KUKA KRL program: MyProgram_247().src

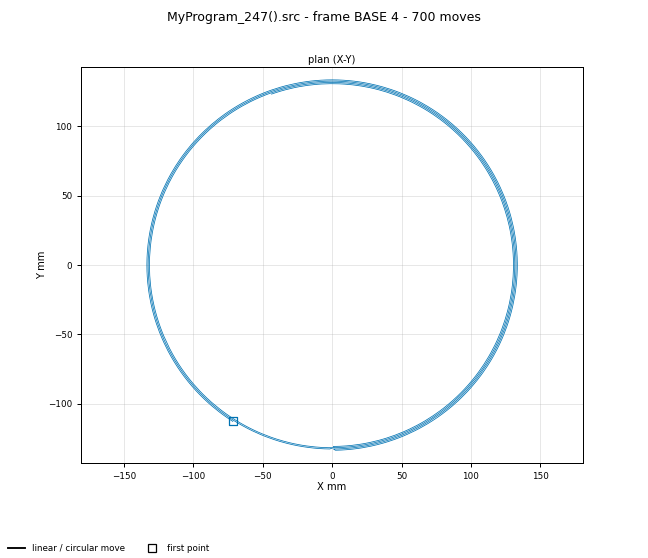
[picture p0: tool path of MyProgram_247().src in frame BASE 4, 700 of 700 moves have a stored position in this frame; points joined in program order, loops and branches not executed]
&ACCESS RVP
&REL 1
&PARAM TEMPLATE = C:\KRC\Roboter\Template\vorgabe
&PARAM EDITMASK = *
DEF MyProgram_247()
; ---- Setting reference (Base) ----
$BASE = BASE_DATA[4]

; --------------------------
; ---- Setting tool (TCP) ----
$TOOL = TOOL_DATA[3]
; --------------------------

$VEL.CP = VEL_APROX_PRINT
Startdeposition()
$VEL.CP = VEL_PRINT
LIN {X -71.493,Y -112.6019,Z 163,A -123.3561,B 17.1544,C -0.1467,E1 17.0685,E2 572.4018} C_DIS
LIN {X -75.0685,Y -110.2504,Z 163,A -125.3445,B 17.1544,C -0.1445,E1 17.0639,E2 574.4076} C_DIS
LIN {X -78.1075,Y -108.1183,Z 163,A -126.8432,B 17.1544,C -0.1504,E1 17.0605,E2 575.894} C_DIS
LIN {X -81.3821,Y -105.6761,Z 163,A -128.5777,B 17.1544,C -0.1541,E1 17.0566,E2 577.6254} C_DIS
LIN {X -86.3277,Y -101.6752,Z 163,A -131.1047,B 17.1542,C -0.166,E1 17.0512,E2 580.1262} C_DIS
LIN {X -88.6867,Y -99.625,Z 163,A -132.7207,B 17.1542,C -0.1593,E1 17.0478,E2 581.7745} C_DIS
LIN {X -91.9669,Y -96.6046,Z 163,A -134.5073,B 17.1542,C -0.1674,E1 17.0442,E2 583.5445} C_DIS
LIN {X -94.7724,Y -93.8538,Z 163,A -136.2946,B 17.1542,C -0.1676,E1 17.0406,E2 585.3427} C_DIS
LIN {X -97.8558,Y -90.6348,Z 163,A -138.7329,B 17.1542,C -0.1544,E1 17.0358,E2 587.8423} C_DIS
LIN {X -100.9904,Y -87.1278,Z 163,A -140.252,B 17.1542,C -0.1754,E1 17.0332,E2 589.3} C_DIS
LIN {X -103.7241,Y -83.8549,Z 163,A -142.1379,B 17.1541,C -0.1777,E1 17.0298,E2 591.1911} C_DIS
LIN {X -106.4808,Y -80.3252,Z 163,A -144.0554,B 17.1541,C -0.1825,E1 17.0265,E2 593.1062} C_DIS
LIN {X -108.9064,Y -77.0047,Z 163,A -145.9648,B 17.1541,C -0.182,E1 17.0234,E2 595.0313} C_DIS
LIN {X -111.3214,Y -73.4702,Z 163,A -147.8571,B 17.1541,C -0.1848,E1 17.0205,E2 596.9283} C_DIS
LIN {X -113.8818,Y -69.4362,Z 163,A -149.7846,B 17.1539,C -0.1941,E1 17.0177,E2 598.8391} C_DIS
LIN {X -116.1067,Y -65.6481,Z 163,A -151.7008,B 17.1539,C -0.198,E1 17.015,E2 600.7569} C_DIS
LIN {X -118.1805,Y -61.8319,Z 163,A -153.4872,B 17.1538,C -0.2055,E1 17.0127,E2 602.5319} C_DIS
LIN {X -121.0994,Y -55.8993,Z 163,A -156.3246,B 17.1537,C -0.2133,E1 17.0092,E2 605.3661} C_DIS
LIN {X -122.6412,Y -52.433,Z 163,A -158.0297,B 17.1537,C -0.2153,E1 17.0073,E2 607.0785} C_DIS
LIN {X -124.4335,Y -48.0231,Z 163,A -160.038,B 17.1536,C -0.2222,E1 17.0052,E2 609.0801} C_DIS
LIN {X -125.5485,Y -45.0269,Z 163,A -161.3821,B 17.1536,C -0.227,E1 17.0039,E2 610.4193} C_DIS
LIN {X -126.5856,Y -42.0228,Z 163,A -162.7229,B 17.1535,C -0.2317,E1 17.0027,E2 611.7555} C_DIS
LIN {X -127.612,Y -38.7951,Z 163,A -164.2281,B 17.1535,C -0.2343,E1 17.0015,E2 613.2651} C_DIS
LIN {X -128.5177,Y -35.6805,Z 163,A -165.6488,B 17.1534,C -0.2375,E1 17.0004,E2 614.6873} C_DIS
LIN {X -129.487,Y -31.9922,Z 163,A -167.8792,B 17.1536,C -0.2233,E1 16.9989,E2 616.986} C_DIS
LIN {X -130.5234,Y -27.4589,Z 163,A -169.4683,B 17.1533,C -0.2423,E1 16.9979,E2 618.5243} C_DIS
LIN {X -131.6134,Y -21.6307,Z 163,A -171.8552,B 17.1531,C -0.2551,E1 16.9968,E2 620.8889} C_DIS
LIN {X -132.1401,Y -18.1495,Z 163,A -174.1734,B 17.1534,C -0.234,E1 16.9959,E2 623.3004} C_DIS
LIN {X -132.774,Y -12.687,Z 163,A -176.0605,B 17.1531,C -0.2562,E1 16.9953,E2 625.1285} C_DIS
LIN {X -133.1204,Y -8.3005,Z 163,A -177.7359,B 17.1529,C -0.2689,E1 16.995,E2 626.7758} C_DIS
LIN {X -133.302,Y -4.5701,Z 163,A -179.3698,B 17.1529,C -0.2728,E1 16.9948,E2 628.4112} C_DIS
LIN {X -133.3812,Y 0.1999,Z 163,A 178.3751,B 17.1529,C -0.2725,E1 16.9948,E2 630.6878} C_DIS
LIN {X -133.2788,Y 5.1658,Z 163,A 176.4508,B 17.1527,C -0.2858,E1 16.9949,E2 632.5843} C_DIS
LIN {X -133.0693,Y 9.1017,Z 163,A 174.457,B 17.1527,C -0.2814,E1 16.9953,E2 634.6113} C_DIS
LIN {X -132.6191,Y 14.2152,Z 163,A 172.1193,B 17.1527,C -0.284,E1 16.9959,E2 636.9614} C_DIS
LIN {X -132.1551,Y 18.0393,Z 163,A 170.7216,B 17.1525,C -0.2972,E1 16.9964,E2 638.3265} C_DIS
LIN {X -131.5675,Y 21.906,Z 163,A 169.1689,B 17.1523,C -0.3064,E1 16.9971,E2 639.8618} C_DIS
LIN {X -130.991,Y 25.1241,Z 163,A 167.6851,B 17.1523,C -0.3081,E1 16.9979,E2 641.3529} C_DIS
LIN {X -129.9919,Y 29.8659,Z 163,A 165.6622,B 17.1521,C -0.3163,E1 16.9991,E2 643.3658} C_DIS
LIN {X -129.2337,Y 32.993,Z 163,A 164.2204,B 17.1521,C -0.3186,E1 17,E2 644.8127} C_DIS
LIN {X -127.6785,Y 38.578,Z 163,A 161.5292,B 17.1521,C -0.3196,E1 17.0021,E2 647.524} C_DIS
LIN {X -126.4721,Y 42.3638,Z 163,A 159.979,B 17.1519,C -0.3297,E1 17.0035,E2 649.0532} C_DIS
LIN {X -125.1164,Y 46.2174,Z 163,A 158.1128,B 17.1519,C -0.3312,E1 17.0052,E2 650.93} C_DIS
LIN {X -122.6784,Y 52.3471,Z 163,A 155.4199,B 17.1516,C -0.344,E1 17.008,E2 653.6022} C_DIS
LIN {X -121.5681,Y 54.8744,Z 163,A 154.0171,B 17.1516,C -0.3404,E1 17.0097,E2 655.0289} C_DIS
LIN {X -118.3417,Y 61.5248,Z 163,A 151.085,B 17.1514,C -0.3571,E1 17.0133,E2 657.9277} C_DIS
LIN {X -116.0256,Y 65.7912,Z 163,A 148.7366,B 17.1514,C -0.3544,E1 17.0164,E2 660.3042} C_DIS
LIN {X -112.7569,Y 71.2474,Z 163,A 146.0518,B 17.1512,C -0.3632,E1 17.0203,E2 662.9795} C_DIS
LIN {X -109.7743,Y 75.763,Z 163,A 143.9098,B 17.151,C -0.3752,E1 17.0236,E2 665.0967} C_DIS
LIN {X -107.8305,Y 78.5046,Z 163,A 142.287,B 17.151,C -0.3731,E1 17.0263,E2 666.7386} C_DIS
LIN {X -105.2804,Y 81.8925,Z 163,A 140.2017,B 17.1511,C -0.3692,E1 17.0299,E2 668.8525} C_DIS
LIN {X -101.3359,Y 86.7267,Z 163,A 137.9244,B 17.1507,C -0.3888,E1 17.0339,E2 671.0787} C_DIS
LIN {X -99.1859,Y 89.177,Z 163,A 135.6773,B 17.1512,C -0.3647,E1 17.0382,E2 673.4232} C_DIS
LIN {X -95.5933,Y 93.018,Z 163,A 133.3776,B 17.1512,C -0.3686,E1 17.0427,E2 675.7246} C_DIS
LIN {X -91.7673,Y 96.7945,Z 163,A 131.9655,B 17.1504,C -0.4029,E1 17.0453,E2 677.0286} C_DIS
LIN {X -86.6154,Y 101.4291,Z 163,A 128.4729,B 17.1506,C -0.3923,E1 17.0527,E2 680.5781} C_DIS
LIN {X -84.0592,Y 103.5591,Z 163,A 127.3266,B 17.1503,C -0.4045,E1 17.0551,E2 681.6894} C_DIS
LIN {X -81.7259,Y 105.4096,Z 163,A 125.9695,B 17.1503,C -0.4045,E1 17.0581,E2 683.0541} C_DIS
LIN {X -77.298,Y 108.6989,Z 163,A 123.7781,B 17.1501,C -0.4149,E1 17.063,E2 685.2217} C_DIS
LIN {X -74.477,Y 110.6508,Z 163,A 122.1784,B 17.1501,C -0.4134,E1 17.0667,E2 686.8346} C_DIS
LIN {X -71.3132,Y 112.7154,Z 163,A 120.5812,B 17.1501,C -0.4171,E1 17.0705,E2 688.4269} C_DIS
LIN {X -68.2373,Y 114.6036,Z 163,A 118.9103,B 17.1501,C -0.4157,E1 17.0745,E2 690.1103} C_DIS
LIN {X -64.4041,Y 116.801,Z 163,A 116.4812,B 17.1504,C -0.4012,E1 17.0806,E2 692.5995} C_DIS
LIN {X -60.2581,Y 118.9908,Z 163,A 114.7353,B 17.1501,C -0.4131,E1 17.0848,E2 694.3119} C_DIS
LIN {X -57.2362,Y 120.4736,Z 163,A 113.5999,B 17.1499,C -0.4256,E1 17.0876,E2 695.4093} C_DIS
LIN {X -53.7854,Y 122.0552,Z 163,A 111.6553,B 17.1501,C -0.4172,E1 17.0926,E2 697.3892} C_DIS
LIN {X -50.7486,Y 123.3486,Z 163,A 110.43,B 17.1499,C -0.4255,E1 17.0957,E2 698.5906} C_DIS
LIN {X -46.8423,Y 124.8824,Z 163,A 108.7335,B 17.1497,C -0.4313,E1 17.1001,E2 700.2728} C_DIS
LIN {X -43.603,Y 126.05,Z 163,A 106.2735,B 17.1504,C -0.4,E1 17.1069,E2 702.8461} C_DIS
LIN {X -37.145,Y 128.1023,Z 163,A 104.3419,B 17.1496,C -0.4359,E1 17.1118,E2 704.6608} C_DIS
LIN {X -33.258,Y 129.1664,Z 163,A 102.5415,B 17.1496,C -0.4351,E1 17.1166,E2 706.4681} C_DIS
LIN {X -26.3839,Y 130.7432,Z 163,A 99.5247,B 17.1496,C -0.4379,E1 17.1249,E2 709.481} C_DIS
LIN {X -22.6279,Y 131.447,Z 163,A 97.7835,B 17.1496,C -0.4355,E1 17.1297,E2 711.2328} C_DIS
LIN {X -18.8702,Y 132.0371,Z 163,A 96.2962,B 17.1495,C -0.4415,E1 17.1337,E2 712.7017} C_DIS
LIN {X -15.3622,Y 132.4918,Z 163,A 94.7327,B 17.1495,C -0.4407,E1 17.1381,E2 714.2695} C_DIS
LIN {X -11.4017,Y 132.8907,Z 163,A 93.0376,B 17.1495,C -0.4419,E1 17.1428,E2 715.9617} C_DIS
LIN {X -8.1027,Y 133.1325,Z 163,A 91.61,B 17.1495,C -0.4422,E1 17.1468,E2 717.3892} C_DIS
LIN {X -4.0439,Y 133.318,Z 163,A 89.8115,B 17.1495,C -0.4407,E1 17.1518,E2 719.1932} C_DIS
LIN {X 0.0154,Y 133.3809,Z 163,A 87.9798,B 17.1495,C -0.4379,E1 17.1569,E2 721.0344} C_DIS
LIN {X 4.194,Y 133.3138,Z 163,A 86.2031,B 17.1495,C -0.4386,E1 17.1619,E2 722.808} C_DIS
LIN {X 8.2626,Y 133.1227,Z 163,A 84.6014,B 17.1495,C -0.4437,E1 17.1663,E2 724.3916} C_DIS
LIN {X 11.8743,Y 132.8508,Z 163,A 82.8734,B 17.1495,C -0.4374,E1 17.1712,E2 726.1393} C_DIS
LIN {X 15.9022,Y 132.4274,Z 163,A 81.2741,B 17.1495,C -0.442,E1 17.1756,E2 727.7215} C_DIS
LIN {X 19.7309,Y 131.913,Z 163,A 79.5121,B 17.1495,C -0.4379,E1 17.1805,E2 729.4952} C_DIS
LIN {X 23.404,Y 131.3093,Z 163,A 78.0206,B 17.1495,C -0.441,E1 17.1845,E2 730.9734} C_DIS
LIN {X 26.981,Y 130.6217,Z 163,A 75.7507,B 17.1501,C -0.4153,E1 17.191,E2 733.3263} C_DIS
LIN {X 32.3107,Y 129.4068,Z 163,A 74.2533,B 17.1494,C -0.4441,E1 17.1948,E2 734.7229} C_DIS
LIN {X 36.0725,Y 128.4081,Z 163,A 72.4271,B 17.1496,C -0.4374,E1 17.1997,E2 736.5672} C_DIS
LIN {X 39.3278,Y 127.449,Z 163,A 70.9977,B 17.1496,C -0.4373,E1 17.2035,E2 737.9932} C_DIS
LIN {X 42.3688,Y 126.4704,Z 163,A 69.6413,B 17.1496,C -0.4367,E1 17.2071,E2 739.3476} C_DIS
LIN {X 45.6944,Y 125.3079,Z 163,A 68.1255,B 17.1496,C -0.4352,E1 17.2111,E2 740.8637} C_DIS
LIN {X 48.7199,Y 124.1626,Z 163,A 66.75,B 17.1496,C -0.4344,E1 17.2147,E2 742.2377} C_DIS
LIN {X 51.816,Y 122.9028,Z 163,A 65.3241,B 17.1496,C -0.4332,E1 17.2184,E2 743.6624} C_DIS
LIN {X 54.7217,Y 121.6364,Z 163,A 63.954,B 17.1497,C -0.4313,E1 17.2219,E2 745.0337} C_DIS
LIN {X 57.9536,Y 120.1308,Z 163,A 62.3008,B 17.1499,C -0.4251,E1 17.2261,E2 746.7017} C_DIS
LIN {X 61.1871,Y 118.5179,Z 163,A 60.8946,B 17.1498,C -0.4284,E1 17.2295,E2 748.0908} C_DIS
LIN {X 63.9805,Y 117.0334,Z 163,A 59.243,B 17.1501,C -0.4158,E1 17.2337,E2 749.7776} C_DIS
LIN {X 68.7879,Y 114.2743,Z 163,A 57.0624,B 17.15,C -0.4197,E1 17.2389,E2 751.9351} C_DIS
LIN {X 72.4699,Y 111.9753,Z 163,A 55.1281,B 17.1501,C -0.4143,E1 17.2435,E2 753.8782} C_DIS
LIN {X 76.0879,Y 109.5488,Z 163,A 53.3455,B 17.1501,C -0.4145,E1 17.2475,E2 755.6509} C_DIS
LIN {X 79.6618,Y 106.9781,Z 163,A 51.4591,B 17.1501,C -0.4114,E1 17.2518,E2 757.5375} C_DIS
LIN {X 83.2162,Y 104.2372,Z 163,A 49.5443,B 17.1503,C -0.4084,E1 17.256,E2 759.4516} C_DIS
LIN {X 86.6973,Y 101.361,Z 163,A 47.5814,B 17.1503,C -0.4039,E1 17.2602,E2 761.4184} C_DIS
LIN {X 90.0715,Y 98.3743,Z 163,A 45.6822,B 17.1504,C -0.4015,E1 17.2641,E2 763.3142} C_DIS
LIN {X 93.2865,Y 95.3308,Z 163,A 43.8058,B 17.1504,C -0.3985,E1 17.2679,E2 765.1888} C_DIS
LIN {X 96.3446,Y 92.2391,Z 163,A 41.9487,B 17.1506,C -0.395,E1 17.2715,E2 767.0458} C_DIS
LIN {X 99.4016,Y 88.9361,Z 163,A 40.0407,B 17.1506,C -0.3917,E1 17.2751,E2 768.952} C_DIS
LIN {X 102.3672,Y 85.5064,Z 163,A 38.0904,B 17.1507,C -0.3872,E1 17.2787,E2 770.9041} C_DIS
LIN {X 105.1727,Y 82.0315,Z 163,A 36.1803,B 17.1508,C -0.3831,E1 17.282,E2 772.8147} C_DIS
LIN {X 108.0905,Y 78.1459,Z 163,A 34.3877,B 17.1507,C -0.3893,E1 17.2849,E2 774.5736} C_DIS
LIN {X 109.735,Y 75.8203,Z 163,A 32.8867,B 17.151,C -0.3757,E1 17.2874,E2 776.1091} C_DIS
LIN {X 112.1364,Y 72.221,Z 163,A 31.0231,B 17.151,C -0.3709,E1 17.2902,E2 777.9748} C_DIS
LIN {X 114.4652,Y 68.4695,Z 163,A 29.1486,B 17.1512,C -0.3669,E1 17.2929,E2 779.8483} C_DIS
LIN {X 116.6388,Y 64.6972,Z 163,A 27.3166,B 17.1512,C -0.3635,E1 17.2954,E2 781.6776} C_DIS
LIN {X 119.3725,Y 59.4986,Z 163,A 24.755,B 17.1514,C -0.3553,E1 17.2987,E2 784.2463} C_DIS
LIN {X 121.0966,Y 55.9054,Z 163,A 23.2334,B 17.1514,C -0.3579,E1 17.3005,E2 785.7466} C_DIS
LIN {X 122.475,Y 52.8174,Z 163,A 21.768,B 17.1514,C -0.3534,E1 17.3022,E2 787.2152} C_DIS
LIN {X 123.7138,Y 49.8466,Z 163,A 20.3661,B 17.1515,C -0.3488,E1 17.3037,E2 788.6209} C_DIS
LIN {X 125.0163,Y 46.4848,Z 163,A 18.8361,B 17.1516,C -0.3451,E1 17.3052,E2 790.1504} C_DIS
LIN {X 126.7022,Y 41.6726,Z 163,A 16.4693,B 17.1519,C -0.3321,E1 17.3073,E2 792.5411} C_DIS
LIN {X 127.9499,Y 37.6655,Z 163,A 14.8838,B 17.1518,C -0.3352,E1 17.3086,E2 794.1024} C_DIS
LIN {X 128.8888,Y 34.3151,Z 163,A 13.3791,B 17.1518,C -0.3304,E1 17.3097,E2 795.6101} C_DIS
LIN {X 130.5446,Y 27.3602,Z 163,A 10.4004,B 17.152,C -0.3248,E1 17.3116,E2 798.5815} C_DIS
LIN {X 131.0616,Y 24.7551,Z 163,A 9.1989,B 17.152,C -0.3191,E1 17.3122,E2 799.7917} C_DIS
LIN {X 131.8029,Y 20.4418,Z 163,A 7.3681,B 17.1522,C -0.3153,E1 17.313,E2 801.619} C_DIS
LIN {X 132.2935,Y 16.9835,Z 163,A 5.9213,B 17.1522,C -0.3129,E1 17.3136,E2 803.0612} C_DIS
LIN {X 132.7376,Y 13.0661,Z 163,A 4.1856,B 17.1523,C -0.3061,E1 17.3141,E2 804.8042} C_DIS
LIN {X 133.0365,Y 9.5509,Z 163,A 2.7026,B 17.1523,C -0.3027,E1 17.3144,E2 806.2854} C_DIS
LIN {X 133.2713,Y 5.3591,Z 163,A 0.8516,B 17.1525,C -0.2953,E1 17.3147,E2 808.1446} C_DIS
LIN {X 133.3772,Y 0.8301,Z 163,A -0.9648,B 17.1525,C -0.2944,E1 17.3147,E2 809.9479} C_DIS
LIN {X 133.3491,Y -2.9015,Z 163,A -2.7829,B 17.1527,C -0.2811,E1 17.3147,E2 811.7944} C_DIS
LIN {X 133.172,Y -7.462,Z 163,A -4.6776,B 17.1527,C -0.2776,E1 17.3144,E2 813.6838} C_DIS
LIN {X 132.8946,Y -11.3554,Z 163,A -6.2039,B 17.1527,C -0.2783,E1 17.3141,E2 815.1942} C_DIS
LIN {X 132.5722,Y -14.651,Z 163,A -7.5931,B 17.1528,C -0.2752,E1 17.3137,E2 816.5814} C_DIS
LIN {X 132.0755,Y -18.6012,Z 163,A -9.3503,B 17.1529,C -0.2681,E1 17.3131,E2 818.3467} C_DIS
LIN {X 131.491,Y -22.3645,Z 163,A -10.9245,B 17.1529,C -0.2655,E1 17.3124,E2 819.9157} C_DIS
LIN {X 130.0759,Y -29.4984,Z 163,A -13.7711,B 17.1529,C -0.2668,E1 17.3108,E2 822.733} C_DIS
LIN {X 129.0527,Y -33.7004,Z 163,A -15.95,B 17.1532,C -0.2487,E1 17.3093,E2 824.9539} C_DIS
LIN {X 128.0391,Y -37.361,Z 163,A -17.5537,B 17.1532,C -0.2449,E1 17.3081,E2 826.5565} C_DIS
LIN {X 126.9864,Y -40.796,Z 163,A -18.9769,B 17.1532,C -0.2449,E1 17.3069,E2 827.9674} C_DIS
LIN {X 125.9675,Y -43.8408,Z 163,A -20.3842,B 17.1533,C -0.2398,E1 17.3056,E2 829.38} C_DIS
LIN {X 124.826,Y -46.9928,Z 163,A -21.7511,B 17.1533,C -0.2384,E1 17.3043,E2 830.7402} C_DIS
LIN {X 123.6614,Y -49.9767,Z 163,A -23.1582,B 17.1534,C -0.2331,E1 17.3029,E2 832.1531} C_DIS
LIN {X 122.3286,Y -53.156,Z 163,A -24.6723,B 17.1535,C -0.2276,E1 17.3012,E2 833.6734} C_DIS
LIN {X 120.529,Y -57.1202,Z 163,A -26.973,B 17.1538,C -0.2056,E1 17.2984,E2 836.0292} C_DIS
LIN {X 118.6252,Y -60.9763,Z 163,A -28.1414,B 17.1535,C -0.2266,E1 17.297,E2 837.1176} C_DIS
LIN {X 116.3629,Y -65.1922,Z 163,A -30.2966,B 17.1536,C -0.217,E1 17.2942,E2 839.2881} C_DIS
LIN {X 114.4383,Y -68.5147,Z 163,A -32.0816,B 17.1538,C -0.2072,E1 17.2916,E2 841.0921} C_DIS
LIN {X 111.9838,Y -72.4567,Z 163,A -34.7078,B 17.1541,C -0.1777,E1 17.2875,E2 843.7977} C_DIS
LIN {X 108.8457,Y -77.0908,Z 163,A -36.1924,B 17.1538,C -0.2066,E1 17.2853,E2 845.174} C_DIS
LIN {X 107.0794,Y -79.5257,Z 163,A -38.1888,B 17.1541,C -0.1763,E1 17.2819,E2 847.258} C_DIS
LIN {X 104.2672,Y -83.1786,Z 163,A -39.7653,B 17.154,C -0.1868,E1 17.2792,E2 848.7882} C_DIS
LIN {X 100.1471,Y -88.0963,Z 163,A -42.449,B 17.154,C -0.1828,E1 17.2743,E2 851.4669} C_DIS
LIN {X 97.187,Y -91.3512,Z 163,A -44.3323,B 17.154,C -0.1785,E1 17.2708,E2 853.352} C_DIS
LIN {X 93.0583,Y -95.5538,Z 163,A -47.0279,B 17.1542,C -0.1665,E1 17.2654,E2 856.071} C_DIS
LIN {X 90.6712,Y -97.822,Z 163,A -47.9557,B 17.154,C -0.1819,E1 17.2636,E2 856.9411} C_DIS
LIN {X 86.8093,Y -101.2647,Z 163,A -50.4464,B 17.1542,C -0.1669,E1 17.2583,E2 859.4675} C_DIS
LIN {X 82.6931,Y -104.6526,Z 163,A -53.1213,B 17.1544,C -0.1476,E1 17.2524,E2 862.1921} C_DIS
LIN {X 79.2187,Y -107.3071,Z 163,A -54.5595,B 17.1542,C -0.1605,E1 17.2493,E2 863.5792} C_DIS
LIN {X 75.7434,Y -109.7877,Z 163,A -56.7712,B 17.1544,C -0.1428,E1 17.2441,E2 865.839} C_DIS
LIN {X 72.302,Y -112.084,Z 163,A -58.1844,B 17.1544,C -0.1532,E1 17.2409,E2 867.21} C_DIS
LIN {X 68.6071,Y -114.3832,Z 163,A -60.018,B 17.1544,C -0.1513,E1 17.2365,E2 869.0414} C_DIS
LIN {X 63.2632,Y -117.4228,Z 163,A -62.6363,B 17.1544,C -0.1478,E1 17.2302,E2 871.6597} C_DIS
LIN {X 59.8567,Y -119.1952,Z 163,A -64.5342,B 17.1544,C -0.136,E1 17.2254,E2 873.5897} C_DIS
LIN {X 56.7284,Y -120.716,Z 163,A -65.6812,B 17.1544,C -0.1467,E1 17.2226,E2 874.6959} C_DIS
LIN {X 54.1774,Y -121.8798,Z 163,A -66.8721,B 17.1544,C -0.1455,E1 17.2195,E2 875.8863} C_DIS
LIN {X 51.3383,Y -123.1023,Z 163,A -68.2057,B 17.1544,C -0.1435,E1 17.2161,E2 877.2219} C_DIS
LIN {X 48.1656,Y -124.3781,Z 163,A -69.714,B 17.1544,C -0.1402,E1 17.2122,E2 878.7365} C_DIS
LIN {X 44.5567,Y -125.7181,Z 163,A -71.4591,B 17.1544,C -0.1348,E1 17.2076,E2 880.4943} C_DIS
LIN {X 39.6414,Y -127.353,Z 163,A -73.543,B 17.1544,C -0.1375,E1 17.2021,E2 882.563} C_DIS
LIN {X 36.5954,Y -128.2618,Z 163,A -75.4292,B 17.1546,C -0.117,E1 17.1968,E2 884.5136} C_DIS
LIN {X 32.3464,Y -129.3978,Z 163,A -76.8995,B 17.1545,C -0.1306,E1 17.193,E2 885.9346} C_DIS
LIN {X 28.253,Y -130.352,Z 163,A -78.6338,B 17.1545,C -0.1317,E1 17.1883,E2 887.6617} C_DIS
LIN {X 24.7601,Y -131.0606,Z 163,A -80.1063,B 17.1545,C -0.1327,E1 17.1842,E2 889.1282} C_DIS
LIN {X 21.814,Y -131.5828,Z 163,A -81.396,B 17.1545,C -0.1316,E1 17.1807,E2 890.4193} C_DIS
LIN {X 18.6748,Y -132.065,Z 163,A -82.7582,B 17.1545,C -0.1309,E1 17.1769,E2 891.7821} C_DIS
LIN {X 14.6266,Y -132.5748,Z 163,A -84.5987,B 17.1545,C -0.1268,E1 17.1718,E2 893.6346} C_DIS
LIN {X 10.5342,Y -132.964,Z 163,A -86.4015,B 17.1545,C -0.1246,E1 17.1668,E2 895.443} C_DIS
LIN {X 6.5935,Y -133.2158,Z 163,A -87.9976,B 17.1545,C -0.1277,E1 17.1623,E2 897.0278} C_DIS
LIN {X 2.3994,Y -133.3575,Z 163,A -89.8236,B 17.1545,C -0.1264,E1 17.1572,E2 898.8576} C_DIS
LIN {X 2.3994,Y -133.3575,Z 163,A -89.8236,B 17.1545,C -0.1264,E1 17.1572,E2 898.8576} C_DIS
Enddeposition()
LIN {X 0.9252,Y -132.4528,Z 163,A -88.4816,B 12.714,C 0.1927,E1 12.718,E2 898.6293} C_DIS
Startdeposition()
$VEL.CP = VEL_PRINT
LIN {X 4.65,Y -132.3773,Z 163,A -86.7032,B 12.714,C 0.1879,E1 12.7231,E2 896.8298} C_DIS
LIN {X 8.6149,Y -132.1783,Z 163,A -84.9273,B 12.714,C 0.1858,E1 12.728,E2 895.0459} C_DIS
LIN {X 13.043,Y -131.8147,Z 163,A -83.1114,B 12.714,C 0.1879,E1 12.7331,E2 893.2417} C_DIS
LIN {X 16.933,Y -131.3713,Z 163,A -81.3857,B 12.714,C 0.1862,E1 12.7379,E2 891.5112} C_DIS
LIN {X 20.7774,Y -130.8191,Z 163,A -79.6446,B 12.7141,C 0.1835,E1 12.7427,E2 889.7615} C_DIS
LIN {X 24.735,Y -130.1278,Z 163,A -78.0449,B 12.7141,C 0.1861,E1 12.747,E2 888.1775} C_DIS
LIN {X 27.8978,Y -129.4865,Z 163,A -76.6131,B 12.7141,C 0.1841,E1 12.751,E2 886.7403} C_DIS
LIN {X 31.8651,Y -128.5698,Z 163,A -74.1973,B 12.7144,C 0.1644,E1 12.7578,E2 884.2427} C_DIS
LIN {X 36.8579,Y -127.2268,Z 163,A -72.8328,B 12.7141,C 0.1866,E1 12.7611,E2 882.9837} C_DIS
LIN {X 40.5932,Y -126.0845,Z 163,A -70.9607,B 12.7141,C 0.1798,E1 12.7662,E2 881.088} C_DIS
LIN {X 44.0819,Y -124.9093,Z 163,A -69.292,B 12.7142,C 0.176,E1 12.7706,E2 879.4087} C_DIS
LIN {X 48.0926,Y -123.4184,Z 163,A -67.5243,B 12.7142,C 0.176,E1 12.7752,E2 877.6495} C_DIS
LIN {X 51.8287,Y -121.8992,Z 163,A -65.7247,B 12.7142,C 0.1723,E1 12.7799,E2 875.8418} C_DIS
LIN {X 55.3976,Y -120.3168,Z 163,A -64.3685,B 12.7142,C 0.1794,E1 12.7832,E2 874.5246} C_DIS
LIN {X 61.0215,Y -117.5659,Z 163,A -60.6564,B 12.7146,C 0.1469,E1 12.7928,E2 870.6866} C_DIS
LIN {X 66.1056,Y -114.7852,Z 163,A -58.8364,B 12.7144,C 0.1627,E1 12.797,E2 868.949} C_DIS
LIN {X 69.5157,Y -112.7526,Z 163,A -57.1776,B 12.7144,C 0.1615,E1 12.801,E2 867.2957} C_DIS
LIN {X 77.6184,Y -107.3354,Z 163,A -52.9856,B 12.7144,C 0.1547,E1 12.8107,E2 863.1026} C_DIS
LIN {X 79.9123,Y -105.6387,Z 163,A -51.4002,B 12.7146,C 0.1422,E1 12.8143,E2 861.4726} C_DIS
LIN {X 83.0042,Y -103.2271,Z 163,A -50.2306,B 12.7145,C 0.1542,E1 12.8167,E2 860.366} C_DIS
LIN {X 86.6021,Y -100.2278,Z 163,A -48.0441,B 12.7145,C 0.1454,E1 12.8214,E2 858.1576} C_DIS
LIN {X 89.442,Y -97.7021,Z 163,A -45.8817,B 12.7148,C 0.1269,E1 12.826,E2 855.9296} C_DIS
LIN {X 93.0322,Y -94.29,Z 163,A -44.3094,B 12.7147,C 0.1389,E1 12.829,E2 854.4252} C_DIS
LIN {X 96.812,Y -90.4044,Z 163,A -41.9462,B 12.7147,C 0.1331,E1 12.8336,E2 852.0571} C_DIS
LIN {X 99.0129,Y -87.9889,Z 163,A -39.868,B 12.7149,C 0.1103,E1 12.8376,E2 849.8952} C_DIS
LIN {X 102.7772,Y -83.561,Z 163,A -38.3365,B 12.7147,C 0.1333,E1 12.8401,E2 848.4819} C_DIS
LIN {X 104.5434,Y -81.3394,Z 163,A -36.5214,B 12.7149,C 0.113,E1 12.8433,E2 846.5932} C_DIS
LIN {X 106.9368,Y -78.1672,Z 163,A -35.1598,B 12.7149,C 0.1193,E1 12.8455,E2 845.2735} C_DIS
LIN {X 111.7951,Y -71.0459,Z 163,A -31.4795,B 12.7149,C 0.1114,E1 12.8512,E2 841.5949} C_DIS
LIN {X 114.0314,Y -67.3978,Z 163,A -29.6337,B 12.7149,C 0.1067,E1 12.8539,E2 839.7475} C_DIS
LIN {X 115.9202,Y -64.0937,Z 163,A -27.7268,B 12.7151,C 0.0946,E1 12.8565,E2 837.8066} C_DIS
LIN {X 117.6362,Y -60.8876,Z 163,A -26.5258,B 12.7151,C 0.1014,E1 12.858,E2 836.6493} C_DIS
LIN {X 120.0623,Y -55.9478,Z 163,A -24.1864,B 12.7151,C 0.0961,E1 12.8609,E2 834.3121} C_DIS
LIN {X 121.4879,Y -52.78,Z 163,A -22.7613,B 12.7151,C 0.0942,E1 12.8625,E2 832.8946} C_DIS
LIN {X 122.7392,Y -49.8012,Z 163,A -21.4109,B 12.7151,C 0.0917,E1 12.8639,E2 831.5482} C_DIS
LIN {X 123.8897,Y -46.867,Z 163,A -19.9341,B 12.7151,C 0.0845,E1 12.8654,E2 830.0559} C_DIS
LIN {X 125.0887,Y -43.5644,Z 163,A -18.4302,B 12.7151,C 0.0807,E1 12.8668,E2 828.5522} C_DIS
LIN {X 126.1966,Y -40.2422,Z 163,A -16.9364,B 12.7151,C 0.077,E1 12.8681,E2 827.0591} C_DIS
LIN {X 127.3419,Y -36.4623,Z 163,A -15.1507,B 12.7152,C 0.0697,E1 12.8695,E2 825.2619} C_DIS
LIN {X 128.351,Y -32.7272,Z 163,A -13.6612,B 12.7152,C 0.0704,E1 12.8705,E2 823.7928} C_DIS
LIN {X 129.8568,Y -26.1202,Z 163,A -10.7284,B 12.7152,C 0.0618,E1 12.8723,E2 820.8565} C_DIS
LIN {X 130.6013,Y -22.1011,Z 163,A -8.9604,B 12.7152,C 0.0566,E1 12.8732,E2 819.0863} C_DIS
LIN {X 131.1939,Y -18.2611,Z 163,A -7.1977,B 12.7153,C 0.0491,E1 12.8739,E2 817.3117} C_DIS
LIN {X 131.7029,Y -14.1219,Z 163,A -5.5797,B 12.7153,C 0.0493,E1 12.8744,E2 815.7142} C_DIS
LIN {X 132.0106,Y -10.8795,Z 163,A -4.043,B 12.7153,C 0.0413,E1 12.8748,E2 814.1604} C_DIS
LIN {X 132.2761,Y -6.9447,Z 163,A -2.4321,B 12.7153,C 0.0391,E1 12.875,E2 812.559} C_DIS
LIN {X 132.4304,Y -2.7627,Z 163,A -0.5578,B 12.7153,C 0.0318,E1 12.8752,E2 810.6749} C_DIS
LIN {X 132.4517,Y 1.4833,Z 163,A 1.296,B 12.7153,C 0.0259,E1 12.8752,E2 808.817} C_DIS
LIN {X 132.3361,Y 5.7074,Z 163,A 3.0736,B 12.7153,C 0.0219,E1 12.875,E2 807.0435} C_DIS
LIN {X 132.0915,Y 9.848,Z 163,A 4.7989,B 12.7153,C 0.0187,E1 12.8747,E2 805.3246} C_DIS
LIN {X 131.7124,Y 14.0336,Z 163,A 6.4926,B 12.7153,C 0.017,E1 12.8742,E2 803.644} C_DIS
LIN {X 131.3276,Y 17.2665,Z 163,A 7.8923,B 12.7153,C 0.0131,E1 12.8737,E2 802.2439} C_DIS
LIN {X 130.8393,Y 20.6471,Z 163,A 9.4762,B 12.7154,C 0.0056,E1 12.873,E2 800.6456} C_DIS
LIN {X 130.1395,Y 24.6741,Z 163,A 11.1431,B 12.7154,C 0.0035,E1 12.8722,E2 798.9891} C_DIS
LIN {X 128.3566,Y 32.7051,Z 163,A 14.7923,B 12.7154,C -0.0094,E1 12.8699,E2 795.3256} C_DIS
LIN {X 126.9678,Y 37.7421,Z 163,A 17.7638,B 12.7154,C -0.0369,E1 12.8675,E2 792.2652} C_DIS
LIN {X 125.0134,Y 43.7817,Z 163,A 19.7259,B 12.7154,C -0.0213,E1 12.8658,E2 790.3963} C_DIS
LIN {X 123.5745,Y 47.691,Z 163,A 21.4127,B 12.7154,C -0.0228,E1 12.8642,E2 788.7218} C_DIS
LIN {X 122.2595,Y 50.9666,Z 163,A 22.8699,B 12.7154,C -0.0249,E1 12.8626,E2 787.2717} C_DIS
LIN {X 120.8602,Y 54.2016,Z 163,A 24.3713,B 12.7154,C -0.0283,E1 12.8609,E2 785.7718} C_DIS
LIN {X 119.7096,Y 56.6991,Z 163,A 26.0355,B 12.7154,C -0.0454,E1 12.8589,E2 784.0493} C_DIS
LIN {X 117.8824,Y 60.4055,Z 163,A 27.4023,B 12.7154,C -0.0377,E1 12.8572,E2 782.732} C_DIS
LIN {X 115.6998,Y 64.4917,Z 163,A 29.396,B 12.7154,C -0.0426,E1 12.8545,E2 780.7381} C_DIS
LIN {X 113.8882,Y 67.6389,Z 163,A 30.9874,B 12.7154,C -0.0471,E1 12.8523,E2 779.1431} C_DIS
LIN {X 111.4568,Y 71.5744,Z 163,A 32.8954,B 12.7154,C -0.0494,E1 12.8495,E2 777.2449} C_DIS
LIN {X 109.5164,Y 74.51,Z 163,A 34.4599,B 12.7153,C -0.0543,E1 12.847,E2 775.6743} C_DIS
LIN {X 106.961,Y 78.1334,Z 163,A 36.3454,B 12.7153,C -0.0579,E1 12.844,E2 773.7914} C_DIS
LIN {X 104.3973,Y 81.5281,Z 163,A 38.1939,B 12.7153,C -0.0623,E1 12.8408,E2 771.9409} C_DIS
LIN {X 101.7273,Y 84.8364,Z 163,A 40.0347,B 12.7153,C -0.0665,E1 12.8375,E2 770.0988} C_DIS
LIN {X 98.8726,Y 88.1464,Z 163,A 41.9101,B 12.7153,C -0.0702,E1 12.8341,E2 768.2243} C_DIS
LIN {X 95.7306,Y 91.5486,Z 163,A 43.8305,B 12.7153,C -0.072,E1 12.8304,E2 766.3128} C_DIS
LIN {X 92.6227,Y 94.6919,Z 163,A 45.6994,B 12.7152,C -0.0747,E1 12.8267,E2 764.4482} C_DIS
LIN {X 89.5531,Y 97.5999,Z 163,A 47.5608,B 12.7152,C -0.0792,E1 12.8229,E2 762.5821} C_DIS
LIN {X 86.1731,Y 100.5973,Z 163,A 49.5073,B 12.7152,C -0.0827,E1 12.8188,E2 760.6358} C_DIS
LIN {X 82.8212,Y 103.3747,Z 163,A 51.4088,B 12.7152,C -0.0867,E1 12.8147,E2 758.7316} C_DIS
LIN {X 79.2848,Y 106.1106,Z 163,A 53.3086,B 12.7151,C -0.0891,E1 12.8105,E2 756.8352} C_DIS
LIN {X 75.6924,Y 108.7021,Z 163,A 55.072,B 12.7151,C -0.0879,E1 12.8065,E2 755.0895} C_DIS
LIN {X 72.9914,Y 110.534,Z 163,A 56.6183,B 12.7151,C -0.0939,E1 12.8029,E2 753.5269} C_DIS
LIN {X 69.0663,Y 113.0283,Z 163,A 58.4818,B 12.7151,C -0.0929,E1 12.7985,E2 751.6807} C_DIS
LIN {X 64.6683,Y 115.601,Z 163,A 60.8194,B 12.7151,C -0.0997,E1 12.7928,E2 749.3268} C_DIS
LIN {X 60.5595,Y 117.804,Z 163,A 62.6476,B 12.7151,C -0.0971,E1 12.7884,E2 747.5208} C_DIS
LIN {X 56.4548,Y 119.8263,Z 163,A 64.7873,B 12.715,C -0.104,E1 12.7829,E2 745.362} C_DIS
LIN {X 52.8847,Y 121.4426,Z 163,A 66.2804,B 12.715,C -0.1004,E1 12.7792,E2 743.8928} C_DIS
LIN {X 49.8992,Y 122.6997,Z 163,A 67.8199,B 12.715,C -0.1056,E1 12.7752,E2 742.3369} C_DIS
LIN {X 46.3379,Y 124.0879,Z 163,A 69.4237,B 12.715,C -0.1059,E1 12.771,E2 740.7391} C_DIS
LIN {X 42.6908,Y 125.3916,Z 163,A 71.2161,B 12.715,C -0.1106,E1 12.7662,E2 738.9329} C_DIS
LIN {X 38.9367,Y 126.6056,Z 163,A 72.965,B 12.715,C -0.1132,E1 12.7616,E2 737.1791} C_DIS
LIN {X 33.5909,Y 128.1288,Z 163,A 74.9974,B 12.715,C -0.1049,E1 12.7562,E2 735.1913} C_DIS
LIN {X 29.7732,Y 129.0683,Z 163,A 77.2376,B 12.7148,C -0.1204,E1 12.75,E2 732.8874} C_DIS
LIN {X 26.2733,Y 129.826,Z 163,A 78.4764,B 12.7149,C -0.1129,E1 12.7467,E2 731.6858} C_DIS
LIN {X 22.0013,Y 130.6179,Z 163,A 80.3225,B 12.7149,C -0.1129,E1 12.7416,E2 729.8442} C_DIS
LIN {X 18.2101,Y 131.2012,Z 163,A 82.0872,B 12.7149,C -0.1163,E1 12.7367,E2 728.0675} C_DIS
LIN {X 14.1813,Y 131.6965,Z 163,A 83.701,B 12.7149,C -0.113,E1 12.7323,E2 726.4711} C_DIS
LIN {X 10.304,Y 132.0582,Z 163,A 85.4447,B 12.7149,C -0.1149,E1 12.7274,E2 724.721} C_DIS
LIN {X 6.735,Y 132.2866,Z 163,A 86.9572,B 12.7149,C -0.1141,E1 12.7232,E2 723.2132} C_DIS
LIN {X 2.7625,Y 132.4304,Z 163,A 88.7321,B 12.7149,C -0.1156,E1 12.7182,E2 721.4326} C_DIS
LIN {X -0.9209,Y 132.455,Z 163,A 90.3145,B 12.7149,C -0.1152,E1 12.7138,E2 719.8522} C_DIS
LIN {X -5.1204,Y 132.359,Z 163,A 92.0701,B 12.7149,C -0.1133,E1 12.7089,E2 718.1047} C_DIS
LIN {X -9.0105,Y 132.1526,Z 163,A 93.8658,B 12.7149,C -0.1158,E1 12.7039,E2 716.2969} C_DIS
LIN {X -13.0008,Y 131.8188,Z 163,A 95.5964,B 12.7149,C -0.1151,E1 12.6991,E2 714.5674} C_DIS
LIN {X -17.4047,Y 131.3095,Z 163,A 97.4277,B 12.7149,C -0.1121,E1 12.694,E2 712.7474} C_DIS
LIN {X -21.4936,Y 130.7026,Z 163,A 99.1645,B 12.7149,C -0.1098,E1 12.6893,E2 711.0179} C_DIS
LIN {X -24.6832,Y 130.1377,Z 163,A 100.6303,B 12.7149,C -0.1106,E1 12.6852,E2 709.5453} C_DIS
LIN {X -34.3405,Y 127.9289,Z 163,A 105.4522,B 12.7149,C -0.121,E1 12.672,E2 704.6631} C_DIS
LIN {X -38.6665,Y 126.6883,Z 163,A 107.3273,B 12.7149,C -0.1173,E1 12.667,E2 702.798} C_DIS
LIN {X -42.6906,Y 125.3916,Z 163,A 108.7765,B 12.7149,C -0.1059,E1 12.6633,E2 701.3954} C_DIS
LIN {X -46.2323,Y 124.1274,Z 163,A 110.3229,B 12.715,C -0.1022,E1 12.6592,E2 699.8597} C_DIS
LIN {X -49.2688,Y 122.9538,Z 163,A 111.6789,B 12.715,C -0.0992,E1 12.6557,E2 698.511} C_DIS
LIN {X -51.5663,Y 122.0091,Z 163,A 112.9535,B 12.715,C -0.1029,E1 12.6524,E2 697.2138} C_DIS
LIN {X -56.2661,Y 119.9152,Z 163,A 115.0618,B 12.715,C -0.0971,E1 12.6471,E2 695.1213} C_DIS
LIN {X -64.3741,Y 115.765,Z 163,A 119.1383,B 12.715,C -0.0947,E1 12.637,E2 691.0327} C_DIS
LIN {X -68.2537,Y 113.5211,Z 163,A 121.109,B 12.715,C -0.0925,E1 12.6322,E2 689.0601} C_DIS
LIN {X -72.1031,Y 111.1154,Z 163,A 122.9055,B 12.7151,C -0.0852,E1 12.628,E2 687.2852} C_DIS
LIN {X -75.3244,Y 108.9582,Z 163,A 124.8645,B 12.7151,C -0.0891,E1 12.6234,E2 685.2946} C_DIS
LIN {X -79.5903,Y 105.8817,Z 163,A 127.0494,B 12.7151,C -0.0828,E1 12.6186,E2 683.1228} C_DIS
LIN {X -83.3142,Y 102.9771,Z 163,A 129.8803,B 12.7151,C -0.098,E1 12.6122,E2 680.2003} C_DIS
LIN {X -88.0879,Y 98.925,Z 163,A 131.8523,B 12.7151,C -0.0747,E1 12.6083,E2 678.319} C_DIS
LIN {X -91.2102,Y 96.054,Z 163,A 133.6127,B 12.7152,C -0.0691,E1 12.6047,E2 676.5694} C_DIS
LIN {X -95.1165,Y 92.1865,Z 163,A 136.3789,B 12.7152,C -0.0732,E1 12.5992,E2 673.7599} C_DIS
LIN {X -97.7163,Y 89.4266,Z 163,A 137.6818,B 12.7152,C -0.0615,E1 12.5968,E2 672.4988} C_DIS
LIN {X -100.4054,Y 86.3958,Z 163,A 139.4473,B 12.7152,C -0.0578,E1 12.5935,E2 670.7338} C_DIS
LIN {X -104.3475,Y 81.5915,Z 163,A 142.2113,B 12.7152,C -0.0533,E1 12.5887,E2 667.964} C_DIS
LIN {X -107.0064,Y 78.0724,Z 163,A 144.1407,B 12.7153,C -0.0491,E1 12.5855,E2 666.0342} C_DIS
LIN {X -109.3849,Y 74.703,Z 163,A 146.2794,B 12.7153,C -0.0531,E1 12.582,E2 663.8556} C_DIS
LIN {X -111.5429,Y 71.44,Z 163,A 147.2842,B 12.7153,C -0.0326,E1 12.5806,E2 662.9341} C_DIS
LIN {X -114.3927,Y 66.7828,Z 163,A 150.0636,B 12.7153,C -0.0362,E1 12.5766,E2 660.1085} C_DIS
LIN {X -116.4876,Y 63.058,Z 163,A 151.8917,B 12.7153,C -0.0309,E1 12.5741,E2 658.2849} C_DIS
LIN {X -119.4398,Y 57.2638,Z 163,A 154.637,B 12.7153,C -0.0217,E1 12.5707,E2 655.5511} C_DIS
LIN {X -120.9308,Y 54.0437,Z 163,A 156.1039,B 12.7153,C -0.016,E1 12.569,E2 654.094} C_DIS
LIN {X -122.3791,Y 50.6804,Z 163,A 157.9599,B 12.7153,C -0.0179,E1 12.5669,E2 652.2078} C_DIS
LIN {X -124.1589,Y 46.1485,Z 163,A 160.0292,B 12.7154,C -0.0111,E1 12.5649,E2 650.1454} C_DIS
LIN {X -125.5479,Y 42.2241,Z 163,A 161.7926,B 12.7154,C -0.0052,E1 12.5633,E2 648.3886} C_DIS
LIN {X -127.4556,Y 36.059,Z 163,A 164.6575,B 12.7154,C 0.0012,E1 12.561,E2 645.5184} C_DIS
LIN {X -128.4866,Y 32.193,Z 163,A 166.3411,B 12.7154,C 0.0073,E1 12.5598,E2 643.8425} C_DIS
LIN {X -129.3249,Y 28.6461,Z 163,A 167.8927,B 12.7154,C 0.0124,E1 12.5588,E2 642.2958} C_DIS
LIN {X -130.0035,Y 25.3852,Z 163,A 169.57,B 12.7154,C 0.0112,E1 12.5579,E2 640.5921} C_DIS
LIN {X -130.8534,Y 20.5558,Z 163,A 171.4685,B 12.7154,C 0.0226,E1 12.557,E2 638.7225} C_DIS
LIN {X -131.7481,Y 13.7022,Z 163,A 174.4909,B 12.7154,C 0.0307,E1 12.556,E2 635.6999} C_DIS
LIN {X -132.2443,Y 7.5445,Z 163,A 177.3597,B 12.7154,C 0.0341,E1 12.5554,E2 632.8109} C_DIS
LIN {X -132.3931,Y 4.1756,Z 163,A 179.2027,B 12.7154,C 0.0295,E1 12.5552,E2 630.9236} C_DIS
LIN {X -132.4614,Y -0.0274,Z 163,A -178.9118,B 12.7154,C 0.0333,E1 12.5552,E2 629.0322} C_DIS
LIN {X -132.3943,Y -4.1328,Z 163,A -177.5267,B 12.7154,C 0.0477,E1 12.5553,E2 627.6957} C_DIS
LIN {X -132.1712,Y -8.7302,Z 163,A -175.0457,B 12.7154,C 0.0421,E1 12.5558,E2 625.1582} C_DIS
LIN {X -131.7932,Y -13.2669,Z 163,A -172.7424,B 12.7154,C 0.0401,E1 12.5564,E2 622.8166} C_DIS
LIN {X -131.0373,Y -19.3565,Z 163,A -170.8172,B 12.7152,C 0.065,E1 12.5572,E2 620.9821} C_DIS
LIN {X -129.4744,Y -27.9538,Z 163,A -166.8219,B 12.7152,C 0.0709,E1 12.5593,E2 616.9648} C_DIS
LIN {X -128.3878,Y -32.5823,Z 163,A -164.9934,B 12.7152,C 0.0821,E1 12.5605,E2 615.1656} C_DIS
LIN {X -127.4349,Y -36.1328,Z 163,A -163.3444,B 12.7152,C 0.0852,E1 12.5617,E2 613.5112} C_DIS
LIN {X -126.334,Y -39.8119,Z 163,A -161.7315,B 12.7151,C 0.091,E1 12.563,E2 611.9056} C_DIS
LIN {X -125.1806,Y -43.2992,Z 163,A -160.1189,B 12.7151,C 0.0948,E1 12.5645,E2 610.2916} C_DIS
LIN {X -124.0508,Y -46.4369,Z 163,A -158.6657,B 12.7151,C 0.0986,E1 12.5659,E2 608.8383} C_DIS
LIN {X -122.9349,Y -49.3157,Z 163,A -157.2687,B 12.7151,C 0.1007,E1 12.5673,E2 607.4351} C_DIS
LIN {X -121.2096,Y -53.4203,Z 163,A -154.8996,B 12.7151,C 0.0954,E1 12.57,E2 605.0144} C_DIS
LIN {X -119.5641,Y -57.0034,Z 163,A -153.4714,B 12.715,C 0.1065,E1 12.5717,E2 603.6209} C_DIS
LIN {X -117.4182,Y -61.3028,Z 163,A -151.5504,B 12.7149,C 0.1156,E1 12.5741,E2 601.7205} C_DIS
LIN {X -115.4169,Y -64.9957,Z 163,A -149.6368,B 12.7149,C 0.1179,E1 12.5767,E2 599.7967} C_DIS
LIN {X -113.16,Y -68.8508,Z 163,A -147.7677,B 12.7149,C 0.1242,E1 12.5793,E2 597.9366} C_DIS
LIN {X -110.7549,Y -72.656,Z 163,A -145.6761,B 12.7148,C 0.1255,E1 12.5825,E2 595.829} C_DIS
LIN {X -107.9348,Y -76.7833,Z 163,A -143.4747,B 12.7148,C 0.1297,E1 12.586,E2 593.6243} C_DIS
LIN {X -105.1935,Y -80.4974,Z 163,A -141.5273,B 12.7147,C 0.1355,E1 12.5893,E2 591.684} C_DIS
LIN {X -102.4497,Y -83.9618,Z 163,A -139.5676,B 12.7147,C 0.1386,E1 12.5927,E2 589.7196} C_DIS
LIN {X -98.6549,Y -88.3895,Z 163,A -136.8353,B 12.7147,C 0.1389,E1 12.5978,E2 586.9632} C_DIS
LIN {X -94.8959,Y -92.4143,Z 163,A -134.5822,B 12.7146,C 0.147,E1 12.6021,E2 584.727} C_DIS
LIN {X -91.7054,Y -95.5807,Z 163,A -132.7076,B 12.7146,C 0.1525,E1 12.6058,E2 582.8617} C_DIS
LIN {X -88.6809,Y -98.3939,Z 163,A -130.8172,B 12.7145,C 0.1534,E1 12.6098,E2 580.9594} C_DIS
LIN {X -83.9601,Y -102.4506,Z 163,A -128.0759,B 12.7145,C 0.1571,E1 12.6156,E2 578.2132} C_DIS
LIN {X -80.2174,Y -105.4076,Z 163,A -126.1678,B 12.7144,C 0.1645,E1 12.6198,E2 576.3246} C_DIS
LIN {X -77.244,Y -107.6054,Z 163,A -124.2211,B 12.7144,C 0.1584,E1 12.6243,E2 574.3361} C_DIS
LIN {X -74.4686,Y -109.5445,Z 163,A -122.9673,B 12.7144,C 0.166,E1 12.6271,E2 573.1082} C_DIS
LIN {X -70.7796,Y -111.9632,Z 163,A -120.8041,B 12.7144,C 0.1624,E1 12.6323,E2 570.9144} C_DIS
LIN {X -67.795,Y -113.7952,Z 163,A -119.6101,B 12.7143,C 0.1726,E1 12.635,E2 569.7597} C_DIS
LIN {X -64.6278,Y -115.6237,Z 163,A -117.9767,B 12.7143,C 0.1735,E1 12.639,E2 568.1203} C_DIS
LIN {X -60.6479,Y -117.759,Z 163,A -115.9847,B 12.7143,C 0.175,E1 12.644,E2 566.1238} C_DIS
LIN {X -57.1962,Y -119.4721,Z 163,A -114.4261,B 12.7142,C 0.1797,E1 12.6478,E2 564.5784} C_DIS
LIN {X -54.268,Y -120.8305,Z 163,A -113.034,B 12.7142,C 0.1813,E1 12.6514,E2 563.1868} C_DIS
LIN {X -51.647,Y -121.9754,Z 163,A -111.673,B 12.7142,C 0.1794,E1 12.6549,E2 561.8108} C_DIS
LIN {X -48.1647,Y -123.3904,Z 163,A -110.0877,B 12.7142,C 0.1821,E1 12.659,E2 560.2304} C_DIS
LIN {X -44.9174,Y -124.6091,Z 163,A -108.6099,B 12.7141,C 0.184,E1 12.6629,E2 558.7552} C_DIS
LIN {X -41.9131,Y -125.6515,Z 163,A -107.1882,B 12.7141,C 0.184,E1 12.6667,E2 557.3278} C_DIS
LIN {X -37.7471,Y -126.9664,Z 163,A -105.281,B 12.7141,C 0.1849,E1 12.6717,E2 555.4183} C_DIS
LIN {X -32.4396,Y -128.424,Z 163,A -102.7793,B 12.7141,C 0.1832,E1 12.6785,E2 552.9013} C_DIS
LIN {X -28.1429,Y -129.4336,Z 163,A -101.0318,B 12.7141,C 0.1884,E1 12.6832,E2 551.1732} C_DIS
LIN {X -24.9966,Y -130.0778,Z 163,A -99.6549,B 12.7141,C 0.1894,E1 12.687,E2 549.7973} C_DIS
LIN {X -21.3547,Y -130.7258,Z 163,A -97.9195,B 12.7141,C 0.1864,E1 12.6918,E2 548.0451} C_DIS
LIN {X -17.2856,Y -131.3251,Z 163,A -96.2226,B 12.7141,C 0.189,E1 12.6965,E2 546.3576} C_DIS
LIN {X -13.09,Y -131.8102,Z 163,A -94.3759,B 12.7141,C 0.1888,E1 12.7016,E2 544.5078} C_DIS
LIN {X -9.4279,Y -132.1221,Z 163,A -92.7722,B 12.7141,C 0.1886,E1 12.7061,E2 542.9018} C_DIS
LIN {X -5.2473,Y -132.354,Z 163,A -91.0553,B 12.714,C 0.1911,E1 12.7109,E2 541.1957} C_DIS
LIN {X -1.6789,Y -132.4484,Z 163,A -89.3706,B 12.714,C 0.1872,E1 12.7156,E2 539.4931} C_DIS
LIN {X -1.6789,Y -132.4484,Z 163,A -89.3706,B 12.714,C 0.1872,E1 12.7156,E2 539.4931} C_DIS
Enddeposition()
LIN {X 0.9224,Y -131.532,Z 163,A -88.9245,B 12.7148,C 0.1974,E1 12.7177,E2 539.0932} C_DIS
Startdeposition()
$VEL.CP = VEL_PRINT
LIN {X -2.8031,Y -131.5087,Z 163,A -90.855,B 12.7147,C 0.2057,E1 12.7122,E2 541.0613} C_DIS
LIN {X -7.5487,Y -131.3213,Z 163,A -92.8272,B 12.7147,C 0.2031,E1 12.7067,E2 543.0229} C_DIS
LIN {X -11.9015,Y -130.9991,Z 163,A -94.6794,B 12.7147,C 0.2017,E1 12.7015,E2 544.87} C_DIS
LIN {X -15.2784,Y -130.6469,Z 163,A -96.1626,B 12.7147,C 0.2015,E1 12.6974,E2 546.3542} C_DIS
LIN {X -18.3651,Y -130.2487,Z 163,A -97.5365,B 12.7147,C 0.2016,E1 12.6936,E2 547.7308} C_DIS
LIN {X -22.2726,Y -129.639,Z 163,A -99.3329,B 12.7147,C 0.2029,E1 12.6886,E2 549.5365} C_DIS
LIN {X -27.0193,Y -128.734,Z 163,A -101.7005,B 12.7147,C 0.2087,E1 12.6821,E2 551.9358} C_DIS
LIN {X -30.4616,Y -127.9615,Z 163,A -103.0518,B 12.7147,C 0.2031,E1 12.6785,E2 553.2655} C_DIS
LIN {X -35.2001,Y -126.7395,Z 163,A -104.9655,B 12.7148,C 0.1962,E1 12.6734,E2 555.1536} C_DIS
LIN {X -40.0775,Y -125.2824,Z 163,A -107.2595,B 12.7148,C 0.1966,E1 12.6672,E2 557.457} C_DIS
LIN {X -43.9864,Y -123.9658,Z 163,A -109.1382,B 12.7148,C 0.1971,E1 12.6622,E2 559.3456} C_DIS
LIN {X -47.6918,Y -122.5861,Z 163,A -110.7333,B 12.7148,C 0.1923,E1 12.6581,E2 560.9256} C_DIS
LIN {X -50.1384,Y -121.6074,Z 163,A -111.807,B 12.7149,C 0.1893,E1 12.6553,E2 561.9906} C_DIS
LIN {X -53.296,Y -120.2564,Z 163,A -113.4281,B 12.7149,C 0.1909,E1 12.6512,E2 563.6265} C_DIS
LIN {X -56.41,Y -118.827,Z 163,A -114.9048,B 12.7149,C 0.1888,E1 12.6474,E2 565.1013} C_DIS
LIN {X -59.665,Y -117.226,Z 163,A -116.2455,B 12.715,C 0.1809,E1 12.6441,E2 566.4134} C_DIS
LIN {X -62.7075,Y -115.6298,Z 163,A -118.1091,B 12.715,C 0.1882,E1 12.6394,E2 568.3206} C_DIS
LIN {X -66.2297,Y -113.6492,Z 163,A -119.8863,B 12.715,C 0.1862,E1 12.6351,E2 570.0996} C_DIS
LIN {X -69.8002,Y -111.4918,Z 163,A -121.7004,B 12.715,C 0.1835,E1 12.6308,E2 571.9131} C_DIS
LIN {X -73.4333,Y -109.1332,Z 163,A -123.5919,B 12.715,C 0.1807,E1 12.6264,E2 573.8047} C_DIS
LIN {X -77.0228,Y -106.6298,Z 163,A -125.5161,B 12.715,C 0.1781,E1 12.622,E2 575.7305} C_DIS
LIN {X -80.5178,Y -104.0157,Z 163,A -127.1746,B 12.7152,C 0.169,E1 12.6184,E2 577.3596} C_DIS
LIN {X -86.7795,Y -98.8524,Z 163,A -130.9365,B 12.7152,C 0.1682,E1 12.6103,E2 581.1474} C_DIS
LIN {X -90.0819,Y -95.8524,Z 163,A -132.9416,B 12.7152,C 0.1659,E1 12.6061,E2 583.159} C_DIS
LIN {X -93.1864,Y -92.8369,Z 163,A -134.8562,B 12.7152,C 0.1629,E1 12.6023,E2 585.0762} C_DIS
LIN {X -95.3953,Y -90.5664,Z 163,A -137.2119,B 12.715,C 0.183,E1 12.5977,E2 587.5455} C_DIS
LIN {X -100.1562,Y -85.2708,Z 163,A -139.12,B 12.7155,C 0.1483,E1 12.5944,E2 589.3122} C_DIS
LIN {X -102.7783,Y -82.0916,Z 163,A -141.1845,B 12.7155,C 0.1507,E1 12.5907,E2 591.4076} C_DIS
LIN {X -105.5108,Y -78.5484,Z 163,A -143.141,B 12.7155,C 0.1464,E1 12.5874,E2 593.3637} C_DIS
LIN {X -108.1414,Y -74.8859,Z 163,A -145.1318,B 12.7155,C 0.1424,E1 12.5842,E2 595.3565} C_DIS
LIN {X -110.5527,Y -71.2786,Z 163,A -147.06,B 12.7155,C 0.1387,E1 12.5812,E2 597.2879} C_DIS
LIN {X -112.8525,Y -67.5778,Z 163,A -148.9603,B 12.7156,C 0.1341,E1 12.5784,E2 599.1871} C_DIS
LIN {X -114.8933,Y -64.0472,Z 163,A -150.7622,B 12.7156,C 0.1302,E1 12.5759,E2 600.9907} C_DIS
LIN {X -117.0282,Y -60.0535,Z 163,A -152.4787,B 12.7158,C 0.1192,E1 12.5738,E2 602.6755} C_DIS
LIN {X -121.0275,Y -51.5242,Z 163,A -156.7411,B 12.7158,C 0.1121,E1 12.5688,E2 606.9537} C_DIS
LIN {X -122.3689,Y -48.2507,Z 163,A -158.3583,B 12.7158,C 0.1097,E1 12.567,E2 608.5784} C_DIS
LIN {X -123.6592,Y -44.8369,Z 163,A -159.9604,B 12.7158,C 0.1056,E1 12.5655,E2 610.1806} C_DIS
LIN {X -124.9888,Y -40.9884,Z 163,A -161.8404,B 12.7158,C 0.1031,E1 12.5638,E2 612.0715} C_DIS
LIN {X -126.2208,Y -37.0162,Z 163,A -163.6629,B 12.7159,C 0.0983,E1 12.5623,E2 613.8935} C_DIS
LIN {X -127.2306,Y -33.3851,Z 163,A -165.3682,B 12.7159,C 0.0951,E1 12.5611,E2 615.6048} C_DIS
LIN {X -128.0773,Y -29.9769,Z 163,A -166.7686,B 12.716,C 0.0878,E1 12.5602,E2 616.9886} C_DIS
LIN {X -129.1745,Y -24.8173,Z 163,A -169.2078,B 12.716,C 0.0844,E1 12.5588,E2 619.442} C_DIS
LIN {X -129.9172,Y -20.5835,Z 163,A -171.0038,B 12.716,C 0.0772,E1 12.558,E2 621.2272} C_DIS
LIN {X -130.4178,Y -17.1215,Z 163,A -172.4876,B 12.7161,C 0.0718,E1 12.5574,E2 622.7048} C_DIS
LIN {X -130.8059,Y -13.8506,Z 163,A -174.9061,B 12.716,C 0.0897,E1 12.5567,E2 625.2357} C_DIS
LIN {X -131.3179,Y -7.6042,Z 163,A -176.8825,B 12.7161,C 0.0648,E1 12.5563,E2 627.1222} C_DIS
LIN {X -131.539,Y -0.2553,Z 163,A 179.1429,B 12.7161,C 0.0726,E1 12.5561,E2 631.1824} C_DIS
LIN {X -131.4167,Y 5.6501,Z 163,A 177.4688,B 12.7162,C 0.0448,E1 12.5563,E2 632.7497} C_DIS
LIN {X -130.8876,Y 13.0635,Z 163,A 173.4789,B 12.7162,C 0.0521,E1 12.5572,E2 636.8231} C_DIS
LIN {X -130.311,Y 17.9295,Z 163,A 171.8355,B 12.7162,C 0.0348,E1 12.5578,E2 638.4074} C_DIS
LIN {X -129.3536,Y 23.8758,Z 163,A 169.1591,B 12.7162,C 0.0283,E1 12.5591,E2 641.0868} C_DIS
LIN {X -128.6462,Y 27.4261,Z 163,A 167.6343,B 12.7162,C 0.0225,E1 12.5599,E2 642.6037} C_DIS
LIN {X -127.824,Y 31.0318,Z 163,A 166,B 12.7162,C 0.0184,E1 12.561,E2 644.2388} C_DIS
LIN {X -126.8951,Y 34.6432,Z 163,A 164.2691,B 12.7162,C 0.0161,E1 12.5622,E2 645.9802} C_DIS
LIN {X -126.033,Y 37.6579,Z 163,A 162.8026,B 12.7162,C 0.0144,E1 12.5634,E2 647.4567} C_DIS
LIN {X -124.5057,Y 42.4346,Z 163,A 160.7404,B 12.7163,C 0.0055,E1 12.5652,E2 649.5021} C_DIS
LIN {X -123.5057,Y 45.2627,Z 163,A 159.2489,B 12.7163,C 0.006,E1 12.5666,E2 651.0135} C_DIS
LIN {X -121.8046,Y 49.6567,Z 163,A 157.4166,B 12.7163,C -0.0048,E1 12.5685,E2 652.8178} C_DIS
LIN {X -120.1705,Y 53.488,Z 163,A 155.799,B 12.7163,C -0.0142,E1 12.5702,E2 654.4103} C_DIS
LIN {X -118.769,Y 56.5315,Z 163,A 154.3297,B 12.7163,C -0.018,E1 12.572,E2 655.8791} C_DIS
LIN {X -117.3638,Y 59.3942,Z 163,A 152.5263,B 12.7163,C -0.0123,E1 12.5743,E2 657.7288} C_DIS
LIN {X -114.9274,Y 63.9856,Z 163,A 150.3327,B 12.7163,C -0.0199,E1 12.5772,E2 659.9116} C_DIS
LIN {X -112.6158,Y 67.9711,Z 163,A 148.2857,B 12.7163,C -0.0242,E1 12.5801,E2 661.9608} C_DIS
LIN {X -110.147,Y 71.9036,Z 163,A 146.1971,B 12.7163,C -0.0278,E1 12.5832,E2 664.0546} C_DIS
LIN {X -107.8786,Y 75.2636,Z 163,A 144.4767,B 12.7163,C -0.0333,E1 12.5859,E2 665.7678} C_DIS
LIN {X -105.5426,Y 78.5056,Z 163,A 142.7432,B 12.7163,C -0.0377,E1 12.5888,E2 667.4984} C_DIS
LIN {X -103.3046,Y 81.4283,Z 163,A 141.0228,B 12.7163,C -0.0388,E1 12.5918,E2 669.2304} C_DIS
LIN {X -100.4805,Y 84.8893,Z 163,A 139.097,B 12.7163,C -0.0438,E1 12.5952,E2 671.1517} C_DIS
LIN {X -97.6853,Y 88.0915,Z 163,A 137.2207,B 12.7163,C -0.0474,E1 12.5987,E2 673.0287} C_DIS
LIN {X -94.6397,Y 91.355,Z 163,A 135.2244,B 12.7163,C -0.0505,E1 12.6025,E2 675.0288} C_DIS
LIN {X -91.183,Y 94.8061,Z 163,A 133.1072,B 12.7162,C -0.0553,E1 12.6067,E2 677.1425} C_DIS
LIN {X -88.1442,Y 97.6375,Z 163,A 131.3098,B 12.7162,C -0.0593,E1 12.6104,E2 678.9365} C_DIS
LIN {X -83.7984,Y 101.3914,Z 163,A 128.8164,B 12.7162,C -0.0644,E1 12.6157,E2 681.4263} C_DIS
LIN {X -80.3227,Y 104.1669,Z 163,A 126.8719,B 12.7162,C -0.0679,E1 12.62,E2 683.3696} C_DIS
LIN {X -73.911,Y 108.8099,Z 163,A 123.6795,B 12.7161,C -0.0801,E1 12.6272,E2 686.5289} C_DIS
LIN {X -71.1951,Y 110.6062,Z 163,A 121.9194,B 12.7161,C -0.0744,E1 12.6314,E2 688.3272} C_DIS
LIN {X -67.2831,Y 113.0282,Z 163,A 119.9319,B 12.7161,C -0.078,E1 12.6361,E2 690.3107} C_DIS
LIN {X -64.5237,Y 114.6258,Z 163,A 117.708,B 12.7161,C -0.0603,E1 12.6418,E2 692.6287} C_DIS
LIN {X -58.8685,Y 117.6304,Z 163,A 115.6862,B 12.7161,C -0.0825,E1 12.6466,E2 694.5604} C_DIS
LIN {X -55.3745,Y 119.3128,Z 163,A 113.7471,B 12.7161,C -0.0787,E1 12.6515,E2 696.5267} C_DIS
LIN {X -52.0566,Y 120.7973,Z 163,A 112.5474,B 12.716,C -0.09,E1 12.6545,E2 697.6809} C_DIS
LIN {X -48.2507,Y 122.3689,Z 163,A 110.661,B 12.716,C -0.0898,E1 12.6594,E2 699.5766} C_DIS
LIN {X -44.845,Y 123.6562,Z 163,A 108.4884,B 12.716,C -0.0773,E1 12.6653,E2 701.815} C_DIS
LIN {X -40.0996,Y 125.2754,Z 163,A 106.8845,B 12.716,C -0.0936,E1 12.6694,E2 703.3507} C_DIS
LIN {X -35.9275,Y 126.5361,Z 163,A 105.0642,B 12.716,C -0.0972,E1 12.6742,E2 705.1606} C_DIS
LIN {X -33.0024,Y 127.331,Z 163,A 103.6993,B 12.716,C -0.0972,E1 12.6779,E2 706.5297} C_DIS
LIN {X -26.7468,Y 128.7898,Z 163,A 100.8837,B 12.716,C -0.0988,E1 12.6856,E2 709.3454} C_DIS
LIN {X -23.651,Y 129.394,Z 163,A 99.5168,B 12.716,C -0.0998,E1 12.6893,E2 710.7106} C_DIS
LIN {X -20.2091,Y 129.9752,Z 163,A 98.0044,B 12.716,C -0.1008,E1 12.6935,E2 712.221} C_DIS
LIN {X -16.4076,Y 130.5114,Z 163,A 96.1927,B 12.716,C -0.0981,E1 12.6985,E2 714.0478} C_DIS
LIN {X -12.5258,Y 130.9392,Z 163,A 94.6452,B 12.716,C -0.1026,E1 12.7028,E2 715.5765} C_DIS
LIN {X -8.6826,Y 131.2515,Z 163,A 92.8515,B 12.716,C -0.1002,E1 12.7078,E2 717.3826} C_DIS
LIN {X -4.8446,Y 131.4481,Z 163,A 91.1872,B 12.716,C -0.1008,E1 12.7124,E2 719.0449} C_DIS
LIN {X -0.7023,Y 131.5352,Z 163,A 89.5318,B 12.7159,C -0.1048,E1 12.717,E2 720.6821} C_DIS
LIN {X 2.3558,Y 131.5161,Z 163,A 88.0637,B 12.7159,C -0.1013,E1 12.7212,E2 722.1653} C_DIS
LIN {X 6.5915,Y 131.3718,Z 163,A 86.2369,B 12.7159,C -0.1017,E1 12.7263,E2 723.9892} C_DIS
LIN {X 10.7092,Y 131.1008,Z 163,A 84.5595,B 12.7159,C -0.1046,E1 12.7309,E2 725.652} C_DIS
LIN {X 13.9786,Y 130.7921,Z 163,A 83.1723,B 12.7159,C -0.1054,E1 12.7347,E2 727.0336} C_DIS
LIN {X 16.6103,Y 130.4848,Z 163,A 81.8613,B 12.7159,C -0.101,E1 12.7384,E2 728.3625} C_DIS
LIN {X 20.182,Y 129.9794,Z 163,A 80.3275,B 12.7159,C -0.1014,E1 12.7426,E2 729.8914} C_DIS
LIN {X 23.1718,Y 129.4797,Z 163,A 78.6319,B 12.7159,C -0.091,E1 12.7474,E2 731.63} C_DIS
LIN {X 26.9532,Y 128.7478,Z 163,A 77.1035,B 12.7159,C -0.094,E1 12.7515,E2 733.1409} C_DIS
LIN {X 31.9463,Y 127.5991,Z 163,A 75.0732,B 12.7159,C -0.0979,E1 12.757,E2 735.1475} C_DIS
LIN {X 37.116,Y 126.1916,Z 163,A 72.7333,B 12.7159,C -0.096,E1 12.7633,E2 737.4877} C_DIS
LIN {X 40.7278,Y 125.0747,Z 163,A 71.1725,B 12.7159,C -0.0969,E1 12.7674,E2 739.0383} C_DIS
LIN {X 44.4444,Y 123.8007,Z 163,A 69.4759,B 12.7159,C -0.0958,E1 12.7719,E2 740.733} C_DIS
LIN {X 47.4148,Y 122.6938,Z 163,A 68.0862,B 12.7159,C -0.0942,E1 12.7755,E2 742.1237} C_DIS
LIN {X 50.4408,Y 121.4811,Z 163,A 66.6954,B 12.7159,C -0.0935,E1 12.7791,E2 743.5111} C_DIS
LIN {X 53.2422,Y 120.2804,Z 163,A 65.2745,B 12.7159,C -0.0895,E1 12.7828,E2 744.9429} C_DIS
LIN {X 56.0707,Y 118.9891,Z 163,A 63.8386,B 12.716,C -0.0856,E1 12.7864,E2 746.3884} C_DIS
LIN {X 59.1694,Y 117.4783,Z 163,A 62.3848,B 12.716,C -0.085,E1 12.79,E2 747.8367} C_DIS
LIN {X 62.3581,Y 115.8182,Z 163,A 60.8555,B 12.716,C -0.0839,E1 12.7938,E2 749.3619} C_DIS
LIN {X 65.2845,Y 114.1942,Z 163,A 59.4065,B 12.716,C -0.0821,E1 12.7973,E2 750.8101} C_DIS
LIN {X 68.9641,Y 112.0106,Z 163,A 57.5529,B 12.716,C -0.0797,E1 12.8018,E2 752.6629} C_DIS
LIN {X 74.3786,Y 108.4905,Z 163,A 54.7831,B 12.716,C -0.0764,E1 12.8082,E2 755.4283} C_DIS
LIN {X 77.7602,Y 106.0931,Z 163,A 52.9616,B 12.7161,C -0.073,E1 12.8123,E2 757.2521} C_DIS
LIN {X 81.1771,Y 103.502,Z 163,A 51.1427,B 12.7161,C -0.0711,E1 12.8163,E2 759.0658} C_DIS
LIN {X 84.3716,Y 100.9151,Z 163,A 49.3063,B 12.7161,C -0.0665,E1 12.8203,E2 760.9083} C_DIS
LIN {X 87.7636,Y 97.9792,Z 163,A 47.3802,B 12.7161,C -0.0636,E1 12.8243,E2 762.8318} C_DIS
LIN {X 91.0844,Y 94.9004,Z 163,A 45.4207,B 12.7161,C -0.06,E1 12.8283,E2 764.7906} C_DIS
LIN {X 94.1943,Y 91.8148,Z 163,A 43.533,B 12.7161,C -0.0567,E1 12.832,E2 766.6768} C_DIS
LIN {X 96.9849,Y 88.8614,Z 163,A 41.7818,B 12.7161,C -0.0535,E1 12.8354,E2 768.4267} C_DIS
LIN {X 99.9503,Y 85.5131,Z 163,A 39.817,B 12.7162,C -0.0487,E1 12.839,E2 770.3944} C_DIS
LIN {X 102.7444,Y 82.1342,Z 163,A 37.96,B 12.7162,C -0.0459,E1 12.8422,E2 772.2464} C_DIS
LIN {X 105.3433,Y 78.7733,Z 163,A 35.6747,B 12.7162,C -0.0294,E1 12.8462,E2 774.5836} C_DIS
LIN {X 107.967,Y 75.1365,Z 163,A 34.1092,B 12.7162,C -0.0357,E1 12.8486,E2 776.105} C_DIS
LIN {X 110.6477,Y 71.1304,Z 163,A 32.1359,B 12.7162,C -0.0341,E1 12.8516,E2 778.0649} C_DIS
LIN {X 112.8066,Y 67.6548,Z 163,A 30.3401,B 12.7162,C -0.0293,E1 12.8542,E2 779.8635} C_DIS
LIN {X 114.7594,Y 64.2859,Z 163,A 28.6624,B 12.7162,C -0.0255,E1 12.8565,E2 781.5404} C_DIS
LIN {X 116.9457,Y 60.2155,Z 163,A 26.6531,B 12.7162,C -0.0204,E1 12.8592,E2 783.5508} C_DIS
LIN {X 119.0544,Y 55.9335,Z 163,A 24.5476,B 12.7163,C -0.0142,E1 12.8617,E2 785.661} C_DIS
LIN {X 120.6878,Y 52.31,Z 163,A 22.9957,B 12.7163,C -0.0147,E1 12.8634,E2 787.1931} C_DIS
LIN {X 122.2238,Y 48.6166,Z 163,A 21.1411,B 12.7163,C -0.0067,E1 12.8654,E2 789.0625} C_DIS
LIN {X 123.7567,Y 44.5663,Z 163,A 19.4432,B 12.7163,C -0.007,E1 12.867,E2 790.7397} C_DIS
LIN {X 125.9447,Y 37.9494,Z 163,A 16.364,B 12.7163,C 0.0028,E1 12.8697,E2 793.827} C_DIS
LIN {X 127.0438,Y 34.0853,Z 163,A 14.6146,B 12.7163,C 0.0077,E1 12.871,E2 795.578} C_DIS
LIN {X 127.8503,Y 30.9227,Z 163,A 12.6575,B 12.7163,C 0.0273,E1 12.8723,E2 797.5995} C_DIS
LIN {X 128.91,Y 26.1561,Z 163,A 11.1281,B 12.7163,C 0.0161,E1 12.8732,E2 799.0607} C_DIS
LIN {X 129.6899,Y 21.9678,Z 163,A 9.3194,B 12.7163,C 0.0202,E1 12.8741,E2 800.8658} C_DIS
LIN {X 130.2132,Y 18.6137,Z 163,A 8.0296,B 12.7163,C 0.019,E1 12.8746,E2 802.1346} C_DIS
LIN {X 130.543,Y 16.1501,Z 163,A 6.7718,B 12.7163,C 0.0273,E1 12.875,E2 803.4144} C_DIS
LIN {X 130.8916,Y 13.0222,Z 163,A 5.4347,B 12.7163,C 0.0303,E1 12.8754,E2 804.7489} C_DIS
LIN {X 131.196,Y 9.4653,Z 163,A 3.8861,B 12.7163,C 0.0347,E1 12.8758,E2 806.2984} C_DIS
LIN {X 131.4108,Y 5.8021,Z 163,A 2.1607,B 12.7163,C 0.0432,E1 12.876,E2 808.0407} C_DIS
LIN {X 131.5277,Y 1.6599,Z 163,A 0.6009,B 12.7163,C 0.0414,E1 12.8761,E2 809.5733} C_DIS
LIN {X 131.5194,Y -2.1579,Z 163,A -1.127,B 12.7163,C 0.0482,E1 12.8761,E2 811.3108} C_DIS
LIN {X 131.3844,Y -6.3406,Z 163,A -2.9768,B 12.7162,C 0.0544,E1 12.8759,E2 813.1658} C_DIS
LIN {X 131.106,Y -10.6481,Z 163,A -4.7737,B 12.7162,C 0.0576,E1 12.8755,E2 814.955} C_DIS
LIN {X 130.7837,Y -14.0569,Z 163,A -6.2486,B 12.7162,C 0.0615,E1 12.8751,E2 816.4297} C_DIS
LIN {X 130.273,Y -18.1957,Z 163,A -8.0675,B 12.7162,C 0.067,E1 12.8744,E2 818.251} C_DIS
LIN {X 129.7193,Y -21.7914,Z 163,A -9.9468,B 12.7161,C 0.0802,E1 12.8736,E2 820.1671} C_DIS
LIN {X 129.0565,Y -25.4344,Z 163,A -12.0368,B 12.7159,C 0.0988,E1 12.8724,E2 822.3154} C_DIS
LIN {X 127.7384,Y -31.3873,Z 163,A -13.6526,B 12.7161,C 0.0763,E1 12.8714,E2 823.8111} C_DIS
LIN {X 126.599,Y -35.7026,Z 163,A -15.8194,B 12.7161,C 0.0885,E1 12.8698,E2 826.0069} C_DIS
LIN {X 125.5015,Y -39.3918,Z 163,A -17.5077,B 12.716,C 0.0937,E1 12.8684,E2 827.6987} C_DIS
LIN {X 124.1981,Y -43.3218,Z 163,A -19.1902,B 12.716,C 0.0953,E1 12.8669,E2 829.3688} C_DIS
LIN {X 122.8182,Y -47.0948,Z 163,A -21.0487,B 12.7159,C 0.1034,E1 12.8651,E2 831.2425} C_DIS
LIN {X 121.3795,Y -50.6841,Z 163,A -22.5569,B 12.7159,C 0.1029,E1 12.8635,E2 832.7316} C_DIS
LIN {X 120.1179,Y -53.6057,Z 163,A -23.9105,B 12.7159,C 0.1058,E1 12.862,E2 834.083} C_DIS
LIN {X 118.5587,Y -56.9717,Z 163,A -25.574,B 12.7159,C 0.1116,E1 12.86,E2 835.7541} C_DIS
LIN {X 116.7887,Y -60.5207,Z 163,A -27.1903,B 12.7159,C 0.1131,E1 12.858,E2 837.3593} C_DIS
LIN {X 115.319,Y -63.2772,Z 163,A -28.725,B 12.7157,C 0.1218,E1 12.8559,E2 838.9165} C_DIS
LIN {X 113.3536,Y -66.7334,Z 163,A -30.3875,B 12.7157,C 0.1243,E1 12.8536,E2 840.5728} C_DIS
LIN {X 111.0206,Y -70.5475,Z 163,A -32.059,B 12.7157,C 0.1214,E1 12.8512,E2 842.2135} C_DIS
LIN {X 108.6889,Y -74.0895,Z 163,A -34.1165,B 12.7157,C 0.1322,E1 12.848,E2 844.2985} C_DIS
LIN {X 106.4209,Y -77.3109,Z 163,A -35.7711,B 12.7157,C 0.1347,E1 12.8453,E2 845.9478} C_DIS
LIN {X 103.2623,Y -81.4821,Z 163,A -38.135,B 12.7155,C 0.1427,E1 12.8413,E2 848.3246} C_DIS
LIN {X 97.888,Y -87.8654,Z 163,A -41.3671,B 12.7155,C 0.1397,E1 12.8355,E2 851.5126} C_DIS
LIN {X 93.2693,Y -92.7535,Z 163,A -44.1745,B 12.7155,C 0.1428,E1 12.8301,E2 854.3089} C_DIS
LIN {X 88.049,Y -97.7235,Z 163,A -47.6094,B 12.7153,C 0.158,E1 12.8231,E2 857.7831} C_DIS
LIN {X 84.127,Y -101.1193,Z 163,A -50.0408,B 12.7153,C 0.1675,E1 12.8179,E2 860.2376} C_DIS
LIN {X 80.4652,Y -104.0565,Z 163,A -52.0051,B 12.7153,C 0.1691,E1 12.8136,E2 862.1944} C_DIS
LIN {X 77.2651,Y -106.4542,Z 163,A -53.6698,B 12.7152,C 0.1702,E1 12.8098,E2 863.8516} C_DIS
LIN {X 71.9144,Y -110.14,Z 163,A -56.5455,B 12.7152,C 0.1766,E1 12.8032,E2 866.7357} C_DIS
LIN {X 68.2747,Y -112.4322,Z 163,A -58.4129,B 12.7151,C 0.1795,E1 12.7987,E2 868.6043} C_DIS
LIN {X 65.3094,Y -114.18,Z 163,A -60.0686,B 12.715,C 0.1863,E1 12.7947,E2 870.2802} C_DIS
LIN {X 60.4077,Y -116.8479,Z 163,A -62.3633,B 12.715,C 0.1862,E1 12.7891,E2 872.5609} C_DIS
LIN {X 55.8087,Y -119.1121,Z 163,A -64.5358,B 12.715,C 0.1877,E1 12.7836,E2 874.7282} C_DIS
LIN {X 52.3954,Y -120.6508,Z 163,A -66.0281,B 12.715,C 0.186,E1 12.7798,E2 876.2053} C_DIS
LIN {X 49.5856,Y -121.8332,Z 163,A -67.4778,B 12.7149,C 0.191,E1 12.7761,E2 877.6707} C_DIS
LIN {X 46.1518,Y -123.1742,Z 163,A -68.8587,B 12.7149,C 0.1867,E1 12.7725,E2 879.026} C_DIS
LIN {X 43.7867,Y -124.0369,Z 163,A -70.2131,B 12.7149,C 0.1951,E1 12.7689,E2 880.4124} C_DIS
LIN {X 39.2664,Y -125.5407,Z 163,A -72.0807,B 12.7149,C 0.1916,E1 12.764,E2 882.2567} C_DIS
LIN {X 33.9021,Y -127.0927,Z 163,A -74.7219,B 12.7148,C 0.1995,E1 12.7568,E2 884.9248} C_DIS
LIN {X 29.3715,Y -128.2156,Z 163,A -76.6249,B 12.7148,C 0.1977,E1 12.7517,E2 886.8137} C_DIS
LIN {X 25.2044,Y -129.1005,Z 163,A -78.5019,B 12.7148,C 0.1996,E1 12.7465,E2 888.6946} C_DIS
LIN {X 21.4145,Y -129.7822,Z 163,A -80.1389,B 12.7148,C 0.1996,E1 12.742,E2 890.3279} C_DIS
LIN {X 17.2874,Y -130.3961,Z 163,A -81.8856,B 12.7148,C 0.1987,E1 12.7372,E2 892.0671} C_DIS
LIN {X 13.8976,Y -130.8008,Z 163,A -83.4379,B 12.7148,C 0.2012,E1 12.7329,E2 893.6282} C_DIS
LIN {X 9.6216,Y -131.1846,Z 163,A -85.2831,B 12.7148,C 0.2012,E1 12.7278,E2 895.4716} C_DIS
LIN {X 5.5109,Y -131.4221,Z 163,A -87.1036,B 12.7148,C 0.2025,E1 12.7227,E2 897.2962} C_DIS
LIN {X 1.5103,Y -131.5302,Z 163,A -88.8941,B 12.7147,C 0.2041,E1 12.7177,E2 899.0932} C_DIS
LIN {X 1.5103,Y -131.5302,Z 163,A -88.8941,B 12.7147,C 0.2041,E1 12.7177,E2 899.0932} C_DIS
Enddeposition()
LIN {X 0.9174,Y -130.6131,Z 163,A -88.8337,B 12.7145,C 0.1879,E1 12.7177,E2 898.9595} C_DIS
Startdeposition()
$VEL.CP = VEL_PRINT
LIN {X 5.642,Y -130.4954,Z 163,A -86.2678,B 12.7147,C 0.1744,E1 12.7249,E2 896.3334} C_DIS
LIN {X 10.1771,Y -130.2207,Z 163,A -84.2053,B 12.7147,C 0.1719,E1 12.7307,E2 894.2615} C_DIS
LIN {X 14.3893,Y -129.8217,Z 163,A -82.5357,B 12.7147,C 0.176,E1 12.7353,E2 892.6132} C_DIS
LIN {X 17.5642,Y -129.431,Z 163,A -81.1378,B 12.7147,C 0.1754,E1 12.7392,E2 891.2152} C_DIS
LIN {X 20.4079,Y -129.0125,Z 163,A -79.8288,B 12.7147,C 0.1734,E1 12.7428,E2 889.8994} C_DIS
LIN {X 23.5667,Y -128.4735,Z 163,A -78.4738,B 12.7147,C 0.1738,E1 12.7465,E2 888.5496} C_DIS
LIN {X 27.044,Y -127.7866,Z 163,A -77.0197,B 12.7147,C 0.1754,E1 12.7505,E2 887.1066} C_DIS
LIN {X 30.1712,Y -127.0842,Z 163,A -75.6509,B 12.7147,C 0.1754,E1 12.7542,E2 885.7412} C_DIS
LIN {X 33.2055,Y -126.3254,Z 163,A -74.2774,B 12.7147,C 0.1741,E1 12.7579,E2 884.3665} C_DIS
LIN {X 35.6343,Y -125.6619,Z 163,A -72.885,B 12.7148,C 0.1652,E1 12.7617,E2 882.9386} C_DIS
LIN {X 39.1272,Y -124.6192,Z 163,A -71.4535,B 12.7148,C 0.1682,E1 12.7655,E2 881.5261} C_DIS
LIN {X 42.1677,Y -123.6235,Z 163,A -70.0576,B 12.7148,C 0.1669,E1 12.7692,E2 880.1299} C_DIS
LIN {X 45.1829,Y -122.5537,Z 163,A -68.6621,B 12.7148,C 0.1655,E1 12.7729,E2 878.7343} C_DIS
LIN {X 48.4924,Y -121.281,Z 163,A -67.1136,B 12.7148,C 0.1638,E1 12.7769,E2 877.1852} C_DIS
LIN {X 51.1282,Y -120.1954,Z 163,A -65.6416,B 12.7149,C 0.1561,E1 12.7807,E2 875.6854} C_DIS
LIN {X 55.5348,Y -118.2241,Z 163,A -63.6589,B 12.7149,C 0.1569,E1 12.7857,E2 873.7171} C_DIS
LIN {X 58.7315,Y -116.6678,Z 163,A -62.2929,B 12.7149,C 0.1601,E1 12.7891,E2 872.373} C_DIS
LIN {X 61.2647,Y -115.3578,Z 163,A -60.9296,B 12.7149,C 0.1551,E1 12.7925,E2 870.995} C_DIS
LIN {X 64.0637,Y -113.8279,Z 163,A -59.5461,B 12.7149,C 0.1533,E1 12.7959,E2 869.6121} C_DIS
LIN {X 67.1474,Y -112.0369,Z 163,A -58.0185,B 12.7149,C 0.1518,E1 12.7996,E2 868.0873} C_DIS
LIN {X 69.8726,Y -110.3576,Z 163,A -56.6256,B 12.715,C 0.1497,E1 12.8029,E2 866.6944} C_DIS
LIN {X 72.5555,Y -108.6124,Z 163,A -55.2692,B 12.715,C 0.1486,E1 12.806,E2 865.3423} C_DIS
LIN {X 75.2166,Y -106.7868,Z 163,A -53.8321,B 12.715,C 0.1455,E1 12.8093,E2 863.9012} C_DIS
LIN {X 77.8062,Y -104.9152,Z 163,A -52.4448,B 12.715,C 0.1433,E1 12.8124,E2 862.5141} C_DIS
LIN {X 80.8419,Y -102.5942,Z 163,A -50.7203,B 12.7151,C 0.1387,E1 12.8163,E2 860.782} C_DIS
LIN {X 84.0693,Y -99.9666,Z 163,A -48.8444,B 12.7151,C 0.1336,E1 12.8203,E2 858.898} C_DIS
LIN {X 87.1253,Y -97.3146,Z 163,A -47.2074,B 12.7151,C 0.1339,E1 12.8237,E2 857.2757} C_DIS
LIN {X 89.9186,Y -94.7404,Z 163,A -45.521,B 12.7152,C 0.1297,E1 12.8272,E2 855.5851} C_DIS
LIN {X 92.7456,Y -91.974,Z 163,A -43.7841,B 12.7152,C 0.1259,E1 12.8306,E2 853.8459} C_DIS
LIN {X 95.5406,Y -89.0671,Z 163,A -42.0658,B 12.7152,C 0.1234,E1 12.8339,E2 852.1317} C_DIS
LIN {X 98.1688,Y -86.1625,Z 163,A -40.2724,B 12.7154,C 0.1173,E1 12.8373,E2 850.3273} C_DIS
LIN {X 100.9365,Y -82.9027,Z 163,A -38.4855,B 12.7154,C 0.1154,E1 12.8404,E2 848.5489} C_DIS
LIN {X 103.3948,Y -79.8155,Z 163,A -36.6863,B 12.7154,C 0.1092,E1 12.8436,E2 846.7395} C_DIS
LIN {X 105.6588,Y -76.7932,Z 163,A -35.1684,B 12.7154,C 0.1092,E1 12.846,E2 845.2363} C_DIS
LIN {X 107.5051,Y -74.187,Z 163,A -33.7883,B 12.7154,C 0.1063,E1 12.8482,E2 843.8571} C_DIS
LIN {X 109.2862,Y -71.5374,Z 163,A -32.3996,B 12.7154,C 0.103,E1 12.8504,E2 842.4681} C_DIS
LIN {X 111.0249,Y -68.8075,Z 163,A -30.9825,B 12.7155,C 0.0994,E1 12.8525,E2 841.0496} C_DIS
LIN {X 112.6758,Y -66.0691,Z 163,A -29.5962,B 12.7155,C 0.0962,E1 12.8545,E2 839.6635} C_DIS
LIN {X 114.4282,Y -62.9861,Z 163,A -28.1095,B 12.7155,C 0.0941,E1 12.8565,E2 838.1833} C_DIS
LIN {X 115.9412,Y -60.1538,Z 163,A -26.6579,B 12.7155,C 0.0891,E1 12.8584,E2 836.7247} C_DIS
LIN {X 117.2269,Y -57.605,Z 163,A -25.3813,B 12.7156,C 0.085,E1 12.86,E2 835.4437} C_DIS
LIN {X 118.7458,Y -54.4065,Z 163,A -23.9213,B 12.7156,C 0.0834,E1 12.8617,E2 833.9929} C_DIS
LIN {X 120.0554,Y -51.4521,Z 163,A -22.4861,B 12.7156,C 0.079,E1 12.8633,E2 832.554} C_DIS
LIN {X 121.1528,Y -48.8103,Z 163,A -21.2483,B 12.7156,C 0.076,E1 12.8646,E2 831.3166} C_DIS
LIN {X 122.432,Y -45.5078,Z 163,A -19.711,B 12.7156,C 0.0721,E1 12.8661,E2 829.7795} C_DIS
LIN {X 123.5111,Y -42.4918,Z 163,A -18.3227,B 12.7157,C 0.0685,E1 12.8674,E2 828.3915} C_DIS
LIN {X 124.5154,Y -39.4522,Z 163,A -16.9352,B 12.7157,C 0.065,E1 12.8686,E2 827.0042} C_DIS
LIN {X 125.4451,Y -36.3883,Z 163,A -15.597,B 12.7157,C 0.0629,E1 12.8697,E2 825.6722} C_DIS
LIN {X 126.2993,Y -33.3032,Z 163,A -14.2017,B 12.7157,C 0.0591,E1 12.8707,E2 824.2764} C_DIS
LIN {X 126.9999,Y -30.521,Z 163,A -12.8703,B 12.7157,C 0.0533,E1 12.8716,E2 822.9347} C_DIS
LIN {X 127.7783,Y -27.0826,Z 163,A -11.423,B 12.7157,C 0.0517,E1 12.8724,E2 821.4975} C_DIS
LIN {X 128.3983,Y -23.9728,Z 163,A -10.0214,B 12.7158,C 0.0473,E1 12.8732,E2 820.093} C_DIS
LIN {X 128.8807,Y -21.2216,Z 163,A -8.8089,B 12.7158,C 0.044,E1 12.8737,E2 818.8806} C_DIS
LIN {X 129.3818,Y -17.922,Z 163,A -7.3902,B 12.7158,C 0.0411,E1 12.8743,E2 817.4655} C_DIS
LIN {X 129.7846,Y -14.7328,Z 163,A -5.8497,B 12.7158,C 0.0331,E1 12.8748,E2 815.9079} C_DIS
LIN {X 130.1289,Y -11.2746,Z 163,A -4.524,B 12.7158,C 0.0343,E1 12.8752,E2 814.6041} C_DIS
LIN {X 130.3492,Y -8.3527,Z 163,A -3.11,B 12.7158,C 0.0268,E1 12.8754,E2 813.1733} C_DIS
LIN {X 130.5144,Y -5.1549,Z 163,A -1.7968,B 12.7158,C 0.0253,E1 12.8756,E2 811.8694} C_DIS
LIN {X 130.5944,Y -2.3955,Z 163,A -0.56,B 12.7158,C 0.0209,E1 12.8756,E2 810.6281} C_DIS
LIN {X 130.6076,Y 1.6032,Z 163,A 1.1524,B 12.7158,C 0.0169,E1 12.8756,E2 808.9187} C_DIS
LIN {X 130.528,Y 4.807,Z 163,A 2.5301,B 12.7158,C 0.0136,E1 12.8756,E2 807.5429} C_DIS
LIN {X 130.3495,Y 8.3465,Z 163,A 4.1582,B 12.7158,C 0.0068,E1 12.8753,E2 805.9043} C_DIS
LIN {X 130.0199,Y 12.4647,Z 163,A 5.8497,B 12.7158,C 0.005,E1 12.8749,E2 804.2253} C_DIS
LIN {X 129.6347,Y 15.9893,Z 163,A 7.3755,B 12.7158,C 0.0013,E1 12.8744,E2 802.7014} C_DIS
LIN {X 129.2048,Y 19.1603,Z 163,A 8.7544,B 12.7158,C -0.0021,E1 12.8738,E2 801.324} C_DIS
LIN {X 128.81,Y 21.6452,Z 163,A 9.9042,B 12.7158,C -0.0067,E1 12.8733,E2 800.1676} C_DIS
LIN {X 128.1738,Y 25.1475,Z 163,A 11.3711,B 12.7158,C -0.0084,E1 12.8726,E2 798.7103} C_DIS
LIN {X 127.5114,Y 28.3186,Z 163,A 12.9181,B 12.7158,C -0.0162,E1 12.8716,E2 797.1469} C_DIS
LIN {X 126.6998,Y 31.7459,Z 163,A 14.3419,B 12.7158,C -0.0171,E1 12.8707,E2 795.736} C_DIS
LIN {X 125.9776,Y 34.5055,Z 163,A 15.5382,B 12.7158,C -0.019,E1 12.8698,E2 794.5451} C_DIS
LIN {X 125.0974,Y 37.5711,Z 163,A 16.9595,B 12.7158,C -0.0236,E1 12.8687,E2 793.1198} C_DIS
LIN {X 124.1436,Y 40.6118,Z 163,A 18.3391,B 12.7158,C -0.027,E1 12.8675,E2 791.7411} C_DIS
LIN {X 123.1434,Y 43.5522,Z 163,A 19.7381,B 12.7158,C -0.0319,E1 12.8662,E2 790.3366} C_DIS
LIN {X 122.1524,Y 46.2544,Z 163,A 21.1019,B 12.7158,C -0.0383,E1 12.8649,E2 788.9596} C_DIS
LIN {X 120.6762,Y 49.9785,Z 163,A 22.5429,B 12.7158,C -0.0339,E1 12.8634,E2 787.5546} C_DIS
LIN {X 119.4847,Y 52.7657,Z 163,A 24.045,B 12.7158,C -0.0425,E1 12.8617,E2 786.0311} C_DIS
LIN {X 118.2235,Y 55.5361,Z 163,A 25.4152,B 12.7158,C -0.047,E1 12.8601,E2 784.6556} C_DIS
LIN {X 116.6665,Y 58.7341,Z 163,A 26.774,B 12.7158,C -0.0453,E1 12.8584,E2 783.3194} C_DIS
LIN {X 115.3533,Y 61.2734,Z 163,A 28.1384,B 12.7158,C -0.0517,E1 12.8567,E2 781.941} C_DIS
LIN {X 113.8187,Y 64.0801,Z 163,A 29.5396,B 12.7158,C -0.0552,E1 12.8548,E2 780.539} C_DIS
LIN {X 112.3358,Y 66.6459,Z 163,A 30.8865,B 12.7158,C -0.0599,E1 12.8528,E2 779.1856} C_DIS
LIN {X 110.3611,Y 69.8671,Z 163,A 32.4197,B 12.7158,C -0.0604,E1 12.8506,E2 777.6659} C_DIS
LIN {X 108.605,Y 72.5666,Z 163,A 33.7361,B 12.7158,C -0.0611,E1 12.8486,E2 776.36} C_DIS
LIN {X 106.9756,Y 74.9489,Z 163,A 35.1404,B 12.7158,C -0.0681,E1 12.8463,E2 774.9385} C_DIS
LIN {X 104.4693,Y 78.4043,Z 163,A 37.06,B 12.7157,C -0.0738,E1 12.8431,E2 773.0123} C_DIS
LIN {X 101.9815,Y 81.614,Z 163,A 38.8194,B 12.7157,C -0.0772,E1 12.8401,E2 771.2544} C_DIS
LIN {X 99.545,Y 84.5679,Z 163,A 40.4626,B 12.7157,C -0.0799,E1 12.8371,E2 769.6146} C_DIS
LIN {X 96.6614,Y 87.8495,Z 163,A 42.3711,B 12.7157,C -0.0838,E1 12.8336,E2 767.706} C_DIS
LIN {X 93.6065,Y 91.0983,Z 163,A 44.3209,B 12.7156,C -0.0877,E1 12.8298,E2 765.7561} C_DIS
LIN {X 90.5236,Y 94.1625,Z 163,A 46.2155,B 12.7156,C -0.0912,E1 12.826,E2 763.862} C_DIS
LIN {X 87.2559,Y 97.1977,Z 163,A 48.0588,B 12.7156,C -0.0919,E1 12.8223,E2 762.0312} C_DIS
LIN {X 84.3124,Y 99.7622,Z 163,A 49.7874,B 12.7156,C -0.0955,E1 12.8186,E2 760.3002} C_DIS
LIN {X 81.4792,Y 102.0888,Z 163,A 51.4323,B 12.7156,C -0.0995,E1 12.815,E2 758.6504} C_DIS
LIN {X 78.0865,Y 104.7065,Z 163,A 53.1831,B 12.7156,C -0.0992,E1 12.8112,E2 756.9141} C_DIS
LIN {X 75.496,Y 106.5897,Z 163,A 54.5757,B 12.7155,C -0.1012,E1 12.808,E2 755.5227} C_DIS
LIN {X 72.8624,Y 108.4075,Z 163,A 56.0551,B 12.7155,C -0.1055,E1 12.8046,E2 754.034} C_DIS
LIN {X 69.3943,Y 110.6595,Z 163,A 57.9219,B 12.7155,C -0.1097,E1 12.8001,E2 752.1606} C_DIS
LIN {X 66.0729,Y 112.6736,Z 163,A 59.4765,B 12.7155,C -0.1081,E1 12.7965,E2 750.6233} C_DIS
LIN {X 62.98,Y 114.4316,Z 163,A 60.9742,B 12.7155,C -0.1086,E1 12.7928,E2 749.1327} C_DIS
LIN {X 60.1576,Y 115.9392,Z 163,A 62.4277,B 12.7155,C -0.1118,E1 12.7892,E2 747.6733} C_DIS
LIN {X 57.6069,Y 117.2259,Z 163,A 63.6687,B 12.7154,C -0.1131,E1 12.7861,E2 746.4335} C_DIS
LIN {X 54.8181,Y 118.5555,Z 163,A 65.0362,B 12.7154,C -0.115,E1 12.7827,E2 745.0645} C_DIS
LIN {X 51.4645,Y 120.0501,Z 163,A 66.6221,B 12.7154,C -0.1161,E1 12.7786,E2 743.4815} C_DIS
LIN {X 48.8126,Y 121.1519,Z 163,A 67.8729,B 12.7154,C -0.1172,E1 12.7754,E2 742.2317} C_DIS
LIN {X 45.5096,Y 122.4313,Z 163,A 69.4218,B 12.7154,C -0.1186,E1 12.7713,E2 740.6835} C_DIS
LIN {X 42.4946,Y 123.5102,Z 163,A 70.8205,B 12.7154,C -0.1198,E1 12.7676,E2 739.2855} C_DIS
LIN {X 39.4527,Y 124.5152,Z 163,A 72.2202,B 12.7154,C -0.1208,E1 12.7639,E2 737.8867} C_DIS
LIN {X 36.3906,Y 125.4444,Z 163,A 73.5686,B 12.7154,C -0.1204,E1 12.7603,E2 736.5449} C_DIS
LIN {X 33.8158,Y 126.1626,Z 163,A 74.8313,B 12.7153,C -0.1237,E1 12.7569,E2 735.2719} C_DIS
LIN {X 30.5237,Y 126.9992,Z 163,A 76.3211,B 12.7153,C -0.1246,E1 12.7529,E2 733.7824} C_DIS
LIN {X 27.0768,Y 127.7795,Z 163,A 77.7862,B 12.7153,C -0.1232,E1 12.7489,E2 732.3276} C_DIS
LIN {X 23.9543,Y 128.4019,Z 163,A 79.2066,B 12.7153,C -0.1245,E1 12.745,E2 730.9047} C_DIS
LIN {X 21.1715,Y 128.8891,Z 163,A 80.4289,B 12.7153,C -0.1246,E1 12.7416,E2 729.6847} C_DIS
LIN {X 17.9154,Y 129.3827,Z 163,A 81.8834,B 12.7153,C -0.1254,E1 12.7376,E2 728.2296} C_DIS
LIN {X 14.7416,Y 129.7835,Z 163,A 83.2774,B 12.7153,C -0.1256,E1 12.7338,E2 726.8372} C_DIS
LIN {X 11.2115,Y 130.1342,Z 163,A 84.7612,B 12.7153,C -0.124,E1 12.7297,E2 725.3622} C_DIS
LIN {X 8.661,Y 130.3302,Z 163,A 86.1343,B 12.7153,C -0.1307,E1 12.7258,E2 723.9605} C_DIS
LIN {X 5.1635,Y 130.5141,Z 163,A 87.5127,B 12.7153,C -0.1267,E1 12.722,E2 722.601} C_DIS
LIN {X 1.9491,Y 130.6018,Z 163,A 88.9406,B 12.7153,C -0.1271,E1 12.718,E2 721.1717} C_DIS
LIN {X -1.2547,Y 130.6112,Z 163,A 90.4055,B 12.7153,C -0.1285,E1 12.7139,E2 719.7006} C_DIS
LIN {X -4.6901,Y 130.5325,Z 163,A 91.8728,B 12.7153,C -0.1273,E1 12.7098,E2 718.2387} C_DIS
LIN {X -7.6543,Y 130.3922,Z 163,A 93.2225,B 12.7153,C -0.1282,E1 12.706,E2 716.8841} C_DIS
LIN {X -11.2041,Y 130.1348,Z 163,A 94.6417,B 12.7153,C -0.1241,E1 12.7021,E2 715.4822} C_DIS
LIN {X -14.393,Y 129.8213,Z 163,A 96.0987,B 12.7153,C -0.1249,E1 12.698,E2 714.0201} C_DIS
LIN {X -17.5692,Y 129.4304,Z 163,A 97.5028,B 12.7153,C -0.1243,E1 12.6941,E2 712.6169} C_DIS
LIN {X -20.3974,Y 129.0141,Z 163,A 98.7373,B 12.7153,C -0.1231,E1 12.6907,E2 711.3854} C_DIS
LIN {X -23.57,Y 128.4729,Z 163,A 100.1789,B 12.7153,C -0.1231,E1 12.6868,E2 709.9412} C_DIS
LIN {X -27.0489,Y 127.7855,Z 163,A 101.6396,B 12.7153,C -0.1197,E1 12.6828,E2 708.4926} C_DIS
LIN {X -30.1919,Y 127.0792,Z 163,A 103.167,B 12.7153,C -0.1215,E1 12.6786,E2 706.953} C_DIS
LIN {X -33.2912,Y 126.3025,Z 163,A 104.448,B 12.7153,C -0.1174,E1 12.6752,E2 705.687} C_DIS
LIN {X -37.0436,Y 125.2532,Z 163,A 106.3621,B 12.7153,C -0.1209,E1 12.67,E2 703.7504} C_DIS
LIN {X -40.6114,Y 124.1437,Z 163,A 107.9281,B 12.7153,C -0.1175,E1 12.6659,E2 702.1941} C_DIS
LIN {X -43.622,Y 123.1183,Z 163,A 109.3247,B 12.7153,C -0.1161,E1 12.6622,E2 700.7985} C_DIS
Enddeposition()
END
